LIN {X 0,Y 376.807,Z 677.795,A -85,B 0,C 180,E1 6969.755,E2 6969.755} C_VEL
LIN {X 0,Y 377.916,Z 679.038,A -85,B 0,C 180,E1 6968.251,E2 6968.251} C_VEL
LIN {X 0,Y 381.799,Z 684.185,A -85,B 0,C 180,E1 6963.881,E2 6963.881} C_VEL
LIN {X 0,Y 385.386,Z 689.219,A -85,B 0,C 180,E1 6960.565,E2 6960.565} C_VEL
LIN {X 0,Y 388.333,Z 693.407,A -85,B 0,C 180,E1 6958.19,E2 6958.19} C_VEL
LIN {X 0,Y 368.305,Z 811.662,A -85,B 0,C 180,E1 6956.59,E2 6956.59} C_VEL
LIN {X 0,Y 361.358,Z 842.659,A -85,B 0,C 180,E1 6956.015,E2 6956.015} C_VEL
LIN {X 0,Y 354.554,Z 867.168,A -85,B 0,C 180,E1 6955.437,E2 6955.437} C_VEL
LIN {X 0,Y 345.016,Z 896.006,A -85,B 0,C 180,E1 6954.606,E2 6954.606} C_VEL
LIN {X 0,Y 335.318,Z 920.733,A -85,B 0,C 180,E1 6953.73,E2 6953.73} C_VEL
LIN {X 0,Y 324.822,Z 944.388,A -85,B 0,C 180,E1 6952.726,E2 6952.726} C_VEL
LIN {X 0,Y 311.352,Z 970.875,A -85,B 0,C 180,E1 6951.358,E2 6951.358} C_VEL
LIN {X 0,Y 299.791,Z 991.138,A -85,B 0,C 180,E1 6950.092,E2 6950.092} C_VEL
LIN {X 0,Y 286.197,Z 1012.789,A -85,B 0,C 180,E1 6948.483,E2 6948.483} C_VEL
LIN {X 0,Y 270.48,Z 1035.107,A -85,B 0,C 180,E1 6946.435,E2 6946.435} C_VEL
LIN {X 0,Y 257.169,Z 1052.336,A -85,B 0,C 180,E1 6944.503,E2 6944.503} C_VEL
LIN {X 0,Y 242.609,Z 1069.728,A -85,B 0,C 180,E1 6942.133,E2 6942.133} C_VEL
LIN {X 0,Y 224.581,Z 1089.33,A -85,B 0,C 180,E1 6938.734,E2 6938.734} C_VEL
LIN {X 0,Y 210.449,Z 1103.455,A -85,B 0,C 180,E1 6935.611,E2 6935.611} C_VEL
LIN {X 0,Y 196.681,Z 1116.374,A -85,B 0,C 180,E1 6932.039,E2 6932.039} C_VEL
LIN {X 0,Y 180.199,Z 1130.963,A -85,B 0,C 180,E1 6926.819,E2 6926.819} C_VEL
LIN {X 0,Y 165.985,Z 1142.764,A -85,B 0,C 180,E1 6921.092,E2 6921.092} C_VEL
LIN {X 0,Y 154.943,Z 1151.763,A -85,B 0,C 180,E1 6915.424,E2 6915.424} C_VEL
LIN {X 0,Y 145.332,Z 1159.666,A -85,B 0,C 180,E1 6909.038,E2 6909.038} C_VEL
LIN {X 0,Y 136.611,Z 1167.272,A -85,B 0,C 180,E1 6901.115,E2 6901.115} C_VEL
LIN {X 0,Y 128.839,Z 1175.216,A -85,B 0,C 180,E1 6889.9,E2 6889.9} C_VEL
LIN {X 0,Y 125.403,Z 1180.335,A -85,B 0,C 180,E1 6880.23,E2 6880.23} C_VEL
LIN {X 0,Y 124.293,Z 1183.823,A -85,B 0,C 180,E1 6872.07,E2 6872.07} C_VEL
LIN {X 0,Y 124.366,Z 1186.875,A -85,B 0,C 180,E1 6863.576,E2 6863.576} C_VEL
LIN {X 0,Y 125.855,Z 1189.644,A -85,B 0,C 180,E1 6854.246,E2 6854.246} C_VEL
LIN {X 0,Y 129.594,Z 1191.987,A -85,B 0,C 180,E1 6844.425,E2 6844.425} C_VEL
LIN {X 0,Y 136.729,Z 1193.742,A -85,B 0,C 180,E1 6834.545,E2 6834.545} C_VEL
LIN {X 0,Y 150.578,Z 1194.995,A -85,B 0,C 180,E1 6823.409,E2 6823.409} C_VEL
LIN {X 0,Y 170.241,Z 1195.086,A -85,B 0,C 180,E1 6813.725,E2 6813.725} C_VEL
LIN {X 0,Y 142.996,Z 1208.131,A -85,B 0,C 180,E1 6799.655,E2 6799.655} C_VEL
LIN {X 0,Y 130.919,Z 1215.278,A -85,B 0,C 180,E1 6787.661,E2 6787.661} C_VEL
LIN {X 0,Y 125.246,Z 1219.957,A -85,B 0,C 180,E1 6776.555,E2 6776.555} C_VEL
LIN {X 0,Y 123.484,Z 1223.083,A -85,B 0,C 180,E1 6765.98,E2 6765.98} C_VEL
LIN {X 0,Y 123.974,Z 1224.682,A -85,B 0,C 180,E1 6757.236,E2 6757.236} C_VEL
LIN {X 0,Y 124.697,Z 1225.027,A -85,B 0,C 180,E1 6751.378,E2 6751.378} C_VEL
LIN {X 0,Y 124.597,Z 1224.748,A -85,B 0,C 180,E1 6746.78,E2 6746.78} C_VEL
LIN {X 0,Y 123.843,Z 1223.305,A -85,B 0,C 180,E1 6739.298,E2 6739.298} C_VEL
LIN {X 0,Y 124.209,Z 1220.042,A -85,B 0,C 180,E1 6729.748,E2 6729.748} C_VEL
LIN {X 0,Y 127.003,Z 1215.367,A -85,B 0,C 180,E1 6720.265,E2 6720.265} C_VEL
LIN {X 0,Y 131.824,Z 1209.964,A -85,B 0,C 180,E1 6712.078,E2 6712.078} C_VEL
LIN {X 0,Y 139.062,Z 1203.153,A -85,B 0,C 180,E1 6704.223,E2 6704.223} C_VEL
LIN {X 0,Y 148.239,Z 1195.223,A -85,B 0,C 180,E1 6697.258,E2 6697.258} C_VEL
LIN {X 0,Y 161.017,Z 1184.519,A -85,B 0,C 180,E1 6690.199,E2 6690.199} C_VEL
LIN {X 0,Y 163.262,Z 1182.63,A -85,B 0,C 180,E1 6689.177,E2 6689.177} C_VEL
LIN {X 0,Y 166.713,Z 1178.925,A -85,B 0,C 180,E1 6687.152,E2 6687.152} C_VEL
LIN {X 0,Y 173.816,Z 1168.339,A -85,B 0,C 180,E1 6681.417,E2 6681.417} C_VEL
LIN {X 0,Y 177.356,Z 1164.823,A -85,B 0,C 180,E1 6679.955,E2 6679.955} C_VEL
LIN {X 0,Y 195.152,Z 1148.924,A -85,B 0,C 180,E1 6675.148,E2 6675.148} C_VEL
LIN {X 0,Y 210.446,Z 1134.258,A -85,B 0,C 180,E1 6671.833,E2 6671.833} C_VEL
LIN {X 0,Y 226.878,Z 1117.357,A -85,B 0,C 180,E1 6668.873,E2 6668.873} C_VEL
LIN {X 0,Y 244.954,Z 1096.893,A -85,B 0,C 180,E1 6666.158,E2 6666.158} C_VEL
LIN {X 0,Y 259.21,Z 1079.289,A -85,B 0,C 180,E1 6664.338,E2 6664.338} C_VEL
LIN {X 0,Y 274.75,Z 1058.411,A -85,B 0,C 180,E1 6662.605,E2 6662.605} C_VEL
LIN {X 0,Y 290.515,Z 1034.681,A -85,B 0,C 180,E1 6661.073,E2 6661.073} C_VEL
LIN {X 0,Y 303.162,Z 1013.691,A -85,B 0,C 180,E1 6660,E2 6660} C_VEL
LIN {X 0,Y 317.013,Z 988.12,A -85,B 0,C 180,E1 6658.96,E2 6658.96} C_VEL
LIN {X 0,Y 328.622,Z 963.653,A -85,B 0,C 180,E1 6658.198,E2 6658.198} C_VEL
LIN {X 0,Y 338.703,Z 939.738,A -85,B 0,C 180,E1 6657.608,E2 6657.608} C_VEL
LIN {X 0,Y 348.992,Z 911.206,A -85,B 0,C 180,E1 6657.061,E2 6657.061} C_VEL
LIN {X 0,Y 356.194,Z 886.963,A -85,B 0,C 180,E1 6656.632,E2 6656.632} C_VEL
LIN {X 0,Y 363.113,Z 858.402,A -85,B 0,C 180,E1 6656.162,E2 6656.162} C_VEL
LIN {X 0,Y 372.946,Z 802.823,A -85,B 0,C 180,E1 6655.391,E2 6655.391} C_VEL
LIN {X 0,Y 388.709,Z 710.46,A -85,B 0,C 180,E1 6654.168,E2 6654.168} C_VEL
LIN {X 0,Y 384.521,Z 702.759,A -85,B 0,C 180,E1 6650.722,E2 6650.722} C_VEL
LIN {X 0,Y 380.976,Z 696.51,A -85,B 0,C 180,E1 6647.341,E2 6647.341} C_VEL
LIN {X 0,Y 378.128,Z 691.496,A -85,B 0,C 180,E1 6644.116,E2 6644.116} C_VEL
LIN {X 0,Y 376.181,Z 687.99,A -85,B 0,C 180,E1 6641.56,E2 6641.56} C_VEL
LIN {X 0,Y 374.754,Z 685.841,A -85,B 0,C 180,E1 6639.471,E2 6639.471} C_VEL
LIN {X 0,Y 372.295,Z 683.021,A -85,B 0,C 180,E1 6635.06,E2 6635.06} C_VEL
LIN {X 0,Y 371.245,Z 680.68,A -85,B 0,C 180,E1 6631.879,E2 6631.879} C_VEL
LIN {X 0,Y 370.079,Z 680.013,A -85,B 0,C 180,E1 6626.366,E2 6626.366} C_VEL
LIN {X 0,Y 370.244,Z 680.021,A -85,B 0,C 180,E1 6621.797,E2 6621.797} C_VEL
LIN {X 0,Y 371.851,Z 680.794,A -85,B 0,C 180,E1 6616.285,E2 6616.285} C_VEL
LIN {X 0,Y 374.459,Z 684.922,A -85,B 0,C 180,E1 6610.915,E2 6610.915} C_VEL
LIN {X 0,Y 376.119,Z 686.558,A -85,B 0,C 180,E1 6608.594,E2 6608.594} C_VEL
LIN {X 0,Y 380.047,Z 691.878,A -85,B 0,C 180,E1 6604.083,E2 6604.083} C_VEL
LIN {X 0,Y 383.547,Z 696.823,A -85,B 0,C 180,E1 6600.814,E2 6600.814} C_VEL
LIN {X 0,Y 385.447,Z 699.553,A -85,B 0,C 180,E1 6599.263,E2 6599.263} C_VEL
LIN {X 0,Y 365.956,Z 812.752,A -85,B 0,C 180,E1 6597.777,E2 6597.777} C_VEL
LIN {X 0,Y 358.945,Z 843.602,A -85,B 0,C 180,E1 6597.222,E2 6597.222} C_VEL
LIN {X 0,Y 352.057,Z 868.102,A -85,B 0,C 180,E1 6596.663,E2 6596.663} C_VEL
LIN {X 0,Y 342.867,Z 895.739,A -85,B 0,C 180,E1 6595.897,E2 6595.897} C_VEL
LIN {X 0,Y 332.641,Z 921.554,A -85,B 0,C 180,E1 6595.016,E2 6595.016} C_VEL
LIN {X 0,Y 322.146,Z 944.946,A -85,B 0,C 180,E1 6594.057,E2 6594.057} C_VEL
LIN {X 0,Y 308.801,Z 970.975,A -85,B 0,C 180,E1 6592.764,E2 6592.764} C_VEL
LIN {X 0,Y 296.588,Z 992.136,A -85,B 0,C 180,E1 6591.489,E2 6591.489} C_VEL
LIN {X 0,Y 282.347,Z 1014.496,A -85,B 0,C 180,E1 6589.875,E2 6589.875} C_VEL
LIN {X 0,Y 266.613,Z 1036.422,A -85,B 0,C 180,E1 6587.91,E2 6587.91} C_VEL
LIN {X 0,Y 253.216,Z 1053.48,A -85,B 0,C 180,E1 6586.046,E2 6586.046} C_VEL
LIN {X 0,Y 238.207,Z 1071.101,A -85,B 0,C 180,E1 6583.701,E2 6583.701} C_VEL
LIN {X 0,Y 220.296,Z 1090.178,A -85,B 0,C 180,E1 6580.46,E2 6580.46} C_VEL
LIN {X 0,Y 206.37,Z 1103.827,A -85,B 0,C 180,E1 6577.517,E2 6577.517} C_VEL
LIN {X 0,Y 192.466,Z 1116.606,A -85,B 0,C 180,E1 6574.072,E2 6574.072} C_VEL
LIN {X 0,Y 176.707,Z 1130.265,A -85,B 0,C 180,E1 6569.352,E2 6569.352} C_VEL
LIN {X 0,Y 160.645,Z 1143.256,A -85,B 0,C 180,E1 6563.209,E2 6563.209} C_VEL
LIN {X 0,Y 148.647,Z 1152.69,A -85,B 0,C 180,E1 6557.255,E2 6557.255} C_VEL
LIN {X 0,Y 138.399,Z 1160.788,A -85,B 0,C 180,E1 6550.59,E2 6550.59} C_VEL
LIN {X 0,Y 128.986,Z 1168.636,A -85,B 0,C 180,E1 6542.096,E2 6542.096} C_VEL
LIN {X 0,Y 120.895,Z 1176.564,A -85,B 0,C 180,E1 6530.281,E2 6530.281} C_VEL
LIN {X 0,Y 117.45,Z 1181.552,A -85,B 0,C 180,E1 6520.317,E2 6520.317} C_VEL
LIN {X 0,Y 116.339,Z 1185.131,A -85,B 0,C 180,E1 6511.62,E2 6511.62} C_VEL
LIN {X 0,Y 116.492,Z 1188.213,A -85,B 0,C 180,E1 6502.722,E2 6502.722} C_VEL
LIN {X 0,Y 118.291,Z 1191.127,A -85,B 0,C 180,E1 6492.696,E2 6492.696} C_VEL
LIN {X 0,Y 123.493,Z 1193.867,A -85,B 0,C 180,E1 6480.928,E2 6480.928} C_VEL
LIN {X 0,Y 132.346,Z 1195.748,A -85,B 0,C 180,E1 6470.432,E2 6470.432} C_VEL
LIN {X 0,Y 150.523,Z 1197.202,A -85,B 0,C 180,E1 6458.161,E2 6458.161} C_VEL
LIN {X 0,Y 159.73,Z 1197.368,A -85,B 0,C 180,E1 6453.838,E2 6453.838} C_VEL
LIN {X 0,Y 138.72,Z 1206.55,A -85,B 0,C 180,E1 6443.137,E2 6443.137} C_VEL
LIN {X 0,Y 125.774,Z 1213.147,A -85,B 0,C 180,E1 6431.896,E2 6431.896} C_VEL
LIN {X 0,Y 118.587,Z 1217.907,A -85,B 0,C 180,E1 6420.39,E2 6420.39} C_VEL
LIN {X 0,Y 115.75,Z 1221.168,A -85,B 0,C 180,E1 6409.163,E2 6409.163} C_VEL
LIN {X 0,Y 115.909,Z 1223.037,A -85,B 0,C 180,E1 6398.933,E2 6398.933} C_VEL
LIN {X 0,Y 116.789,Z 1223.531,A -85,B 0,C 180,E1 6391.962,E2 6391.962} C_VEL
LIN {X 0,Y 116.767,Z 1223.202,A -85,B 0,C 180,E1 6387.055,E2 6387.055} C_VEL
LIN {X 0,Y 115.963,Z 1221.726,A -85,B 0,C 180,E1 6379.065,E2 6379.065} C_VEL
LIN {X 0,Y 116.361,Z 1218.627,A -85,B 0,C 180,E1 6369.371,E2 6369.371} C_VEL
LIN {X 0,Y 119.153,Z 1214.237,A -85,B 0,C 180,E1 6359.769,E2 6359.769} C_VEL
LIN {X 0,Y 124.544,Z 1208.555,A -85,B 0,C 180,E1 6350.637,E2 6350.637} C_VEL
LIN {X 0,Y 131.983,Z 1201.99,A -85,B 0,C 180,E1 6342.705,E2 6342.705} C_VEL
LIN {X 0,Y 142.028,Z 1193.772,A -85,B 0,C 180,E1 6335.25,E2 6335.25} C_VEL
LIN {X 0,Y 156.04,Z 1182.615,A -85,B 0,C 180,E1 6327.837,E2 6327.837} C_VEL
LIN {X 0,Y 172.105,Z 1169.246,A -85,B 0,C 180,E1 6321.635,E2 6321.635} C_VEL
LIN {X 0,Y 177.356,Z 1164.823,A -85,B 0,C 180,E1 6319.955,E2 6319.955} C_VEL
LIN {X 0,Y 181.451,Z 1160.675,A -85,B 0,C 180,E1 6318.318,E2 6318.318} C_VEL
LIN {X 0,Y 190.105,Z 1148.761,A -85,B 0,C 180,E1 6313.592,E2 6313.592} C_VEL
LIN {X 0,Y 193.9,Z 1144.78,A -85,B 0,C 180,E1 6312.455,E2 6312.455} C_VEL
LIN {X 0,Y 210.652,Z 1128.923,A -85,B 0,C 180,E1 6309.146,E2 6309.146} C_VEL
LIN {X 0,Y 228.81,Z 1110.021,A -85,B 0,C 180,E1 6306.199,E2 6306.199} C_VEL
LIN {X 0,Y 243.618,Z 1093.246,A -85,B 0,C 180,E1 6304.18,E2 6304.18} C_VEL
LIN {X 0,Y 259.185,Z 1074.103,A -85,B 0,C 180,E1 6302.345,E2 6302.345} C_VEL
LIN {X 0,Y 276.159,Z 1050.89,A -85,B 0,C 180,E1 6300.622,E2 6300.622} C_VEL
LIN {X 0,Y 288.976,Z 1031.521,A -85,B 0,C 180,E1 6299.481,E2 6299.481} C_VEL
LIN {X 0,Y 302.578,Z 1008.982,A -85,B 0,C 180,E1 6298.413,E2 6298.413} C_VEL
LIN {X 0,Y 316.363,Z 983.126,A -85,B 0,C 180,E1 6297.464,E2 6297.464} C_VEL
LIN {X 0,Y 326.962,Z 960.747,A -85,B 0,C 180,E1 6296.821,E2 6296.821} C_VEL
LIN {X 0,Y 338.194,Z 933.985,A -85,B 0,C 180,E1 6296.22,E2 6296.22} C_VEL
LIN {X 0,Y 347.531,Z 907.401,A -85,B 0,C 180,E1 6295.755,E2 6295.755} C_VEL
LIN {X 0,Y 354.672,Z 883.133,A -85,B 0,C 180,E1 6295.345,E2 6295.345} C_VEL
LIN {X 0,Y 361.973,Z 851.727,A -85,B 0,C 180,E1 6294.861,E2 6294.861} C_VEL
LIN {X 0,Y 385.689,Z 715.96,A -85,B 0,C 180,E1 6293.076,E2 6293.076} C_VEL
LIN {X 0,Y 381.393,Z 708.075,A -85,B 0,C 180,E1 6289.349,E2 6289.349} C_VEL
LIN {X 0,Y 378.608,Z 703.267,A -85,B 0,C 180,E1 6286.561,E2 6286.561} C_VEL
LIN {X 0,Y 376.268,Z 699.022,A -85,B 0,C 180,E1 6283.798,E2 6283.798} C_VEL
LIN {X 0,Y 374.464,Z 695.649,A -85,B 0,C 180,E1 6281.311,E2 6281.311} C_VEL
LIN {X 0,Y 373.06,Z 693.606,A -85,B 0,C 180,E1 6279.28,E2 6279.28} C_VEL
LIN {X 0,Y 370.521,Z 690.447,A -85,B 0,C 180,E1 6274.419,E2 6274.419} C_VEL
LIN {X 0,Y 369.676,Z 688.523,A -85,B 0,C 180,E1 6271.853,E2 6271.853} C_VEL
LIN {X 0,Y 368.52,Z 687.86,A -85,B 0,C 180,E1 6266.392,E2 6266.392} C_VEL
LIN {X 0,Y 368.684,Z 687.868,A -85,B 0,C 180,E1 6261.804,E2 6261.804} C_VEL
LIN {X 0,Y 370.35,Z 688.67,A -85,B 0,C 180,E1 6256.17,E2 6256.17} C_VEL
LIN {X 0,Y 372.645,Z 692.538,A -85,B 0,C 180,E1 6251.296,E2 6251.296} C_VEL
LIN {X 0,Y 374.524,Z 694.44,A -85,B 0,C 180,E1 6248.661,E2 6248.661} C_VEL
LIN {X 0,Y 378.327,Z 699.612,A -85,B 0,C 180,E1 6244.259,E2 6244.259} C_VEL
LIN {X 0,Y 381.829,Z 704.599,A -85,B 0,C 180,E1 6240.968,E2 6240.968} C_VEL
LIN {X 0,Y 382.546,Z 705.831,A -85,B 0,C 180,E1 6240.349,E2 6240.349} C_VEL
LIN {X 0,Y 363.729,Z 813.59,A -85,B 0,C 180,E1 6238.979,E2 6238.979} C_VEL
LIN {X 0,Y 356.637,Z 844.412,A -85,B 0,C 180,E1 6238.444,E2 6238.444} C_VEL
LIN {X 0,Y 349.598,Z 869.163,A -85,B 0,C 180,E1 6237.898,E2 6237.898} C_VEL
LIN {X 0,Y 340.237,Z 896.95,A -85,B 0,C 180,E1 6237.155,E2 6237.155} C_VEL
LIN {X 0,Y 329.949,Z 922.634,A -85,B 0,C 180,E1 6236.309,E2 6236.309} C_VEL
LIN {X 0,Y 319.431,Z 945.822,A -85,B 0,C 180,E1 6235.394,E2 6235.394} C_VEL
LIN {X 0,Y 305.662,Z 972.359,A -85,B 0,C 180,E1 6234.122,E2 6234.122} C_VEL
LIN {X 0,Y 293.599,Z 993.014,A -85,B 0,C 180,E1 6232.92,E2 6232.92} C_VEL
LIN {X 0,Y 279.504,Z 1014.888,A -85,B 0,C 180,E1 6231.401,E2 6231.401} C_VEL
LIN {X 0,Y 263.536,Z 1036.941,A -85,B 0,C 180,E1 6229.504,E2 6229.504} C_VEL
LIN {X 0,Y 249.352,Z 1054.743,A -85,B 0,C 180,E1 6227.623,E2 6227.623} C_VEL
LIN {X 0,Y 233.036,Z 1073.544,A -85,B 0,C 180,E1 6225.173,E2 6225.173} C_VEL
LIN {X 0,Y 215.226,Z 1092.006,A -85,B 0,C 180,E1 6222.067,E2 6222.067} C_VEL
LIN {X 0,Y 200.472,Z 1106.103,A -85,B 0,C 180,E1 6219.045,E2 6219.045} C_VEL
LIN {X 0,Y 184.747,Z 1120.107,A -85,B 0,C 180,E1 6215.219,E2 6215.219} C_VEL
LIN {X 0,Y 166.504,Z 1135.133,A -85,B 0,C 180,E1 6209.656,E2 6209.656} C_VEL
LIN {X 0,Y 152.746,Z 1145.818,A -85,B 0,C 180,E1 6204.275,E2 6204.275} C_VEL
LIN {X 0,Y 140.894,Z 1154.778,A -85,B 0,C 180,E1 6198.339,E2 6198.339} C_VEL
LIN {X 0,Y 129.327,Z 1163.597,A -85,B 0,C 180,E1 6190.583,E2 6190.583} C_VEL
LIN {X 0,Y 118.33,Z 1172.568,A -85,B 0,C 180,E1 6179.532,E2 6179.532} C_VEL
LIN {X 0,Y 112.374,Z 1178.516,A -85,B 0,C 180,E1 6169.494,E2 6169.494} C_VEL
LIN {X 0,Y 109.356,Z 1183.037,A -85,B 0,C 180,E1 6159.795,E2 6159.795} C_VEL
LIN {X 0,Y 108.359,Z 1186.606,A -85,B 0,C 180,E1 6150.499,E2 6150.499} C_VEL
LIN {X 0,Y 108.716,Z 1189.747,A -85,B 0,C 180,E1 6141.02,E2 6141.02} C_VEL
LIN {X 0,Y 111.155,Z 1192.843,A -85,B 0,C 180,E1 6129.841,E2 6129.841} C_VEL
LIN {X 0,Y 117.496,Z 1195.665,A -85,B 0,C 180,E1 6117.561,E2 6117.561} C_VEL
LIN {X 0,Y 129.203,Z 1197.861,A -85,B 0,C 180,E1 6105.662,E2 6105.662} C_VEL
LIN {X 0,Y 149.142,Z 1199.417,A -85,B 0,C 180,E1 6093.943,E2 6093.943} C_VEL
LIN {X 0,Y 123.761,Z 1209.945,A -85,B 0,C 180,E1 6078.708,E2 6078.708} C_VEL
LIN {X 0,Y 112.841,Z 1215.61,A -85,B 0,C 180,E1 6065.391,E2 6065.391} C_VEL
LIN {X 0,Y 108.287,Z 1219.269,A -85,B 0,C 180,E1 6052.575,E2 6052.575} C_VEL
LIN {X 0,Y 107.811,Z 1221.319,A -85,B 0,C 180,E1 6041.231,E2 6041.231} C_VEL
LIN {X 0,Y 108.858,Z 1222.015,A -85,B 0,C 180,E1 6032.632,E2 6032.632} C_VEL
LIN {X 0,Y 108.975,Z 1221.736,A -85,B 0,C 180,E1 6027.897,E2 6027.897} C_VEL
LIN {X 0,Y 108.148,Z 1220.405,A -85,B 0,C 180,E1 6019.883,E2 6019.883} C_VEL
LIN {X 0,Y 108.443,Z 1217.37,A -85,B 0,C 180,E1 6009.49,E2 6009.49} C_VEL
LIN {X 0,Y 111.323,Z 1213.03,A -85,B 0,C 180,E1 5999.205,E2 5999.205} C_VEL
LIN {X 0,Y 117,Z 1207.402,A -85,B 0,C 180,E1 5989.496,E2 5989.496} C_VEL
LIN {X 0,Y 124.848,Z 1200.88,A -85,B 0,C 180,E1 5981.164,E2 5981.164} C_VEL
LIN {X 0,Y 134.856,Z 1193.116,A -85,B 0,C 180,E1 5973.786,E2 5973.786} C_VEL
LIN {X 0,Y 147.203,Z 1183.674,A -85,B 0,C 180,E1 5967.149,E2 5967.149} C_VEL
LIN {X 0,Y 165.02,Z 1169.636,A -85,B 0,C 180,E1 5960.205,E2 5960.205} C_VEL
LIN {X 0,Y 179.945,Z 1157.146,A -85,B 0,C 180,E1 5955.8,E2 5955.8} C_VEL
LIN {X 0,Y 193.9,Z 1144.78,A -85,B 0,C 180,E1 5952.455,E2 5952.455} C_VEL
LIN {X 0,Y 198.293,Z 1140.203,A -85,B 0,C 180,E1 5951.164,E2 5951.164} C_VEL
LIN {X 0,Y 207.938,Z 1127.189,A -85,B 0,C 180,E1 5947.266,E2 5947.266} C_VEL
LIN {X 0,Y 211.846,Z 1122.826,A -85,B 0,C 180,E1 5946.393,E2 5946.393} C_VEL
LIN {X 0,Y 227.953,Z 1106.085,A -85,B 0,C 180,E1 5944.024,E2 5944.024} C_VEL
LIN {X 0,Y 244.119,Z 1087.834,A -85,B 0,C 180,E1 5942.007,E2 5942.007} C_VEL
LIN {X 0,Y 261.968,Z 1065.443,A -85,B 0,C 180,E1 5940.112,E2 5940.112} C_VEL
LIN {X 0,Y 276.024,Z 1045.959,A -85,B 0,C 180,E1 5938.822,E2 5938.822} C_VEL
LIN {X 0,Y 291.219,Z 1022.84,A -85,B 0,C 180,E1 5937.603,E2 5937.603} C_VEL
LIN {X 0,Y 305.498,Z 998.135,A -85,B 0,C 180,E1 5936.604,E2 5936.604} C_VEL
LIN {X 0,Y 317.11,Z 975.773,A -85,B 0,C 180,E1 5935.891,E2 5935.891} C_VEL
LIN {X 0,Y 330.437,Z 946.425,A -85,B 0,C 180,E1 5935.177,E2 5935.177} C_VEL
LIN {X 0,Y 339.838,Z 922.429,A -85,B 0,C 180,E1 5934.742,E2 5934.742} C_VEL
LIN {X 0,Y 349.05,Z 894.753,A -85,B 0,C 180,E1 5934.288,E2 5934.288} C_VEL
LIN {X 0,Y 356.298,Z 867.232,A -85,B 0,C 180,E1 5933.866,E2 5933.866} C_VEL
LIN {X 0,Y 361.787,Z 841.172,A -85,B 0,C 180,E1 5933.497,E2 5933.497} C_VEL
LIN {X 0,Y 382.792,Z 721.682,A -85,B 0,C 180,E1 5931.983,E2 5931.983} C_VEL
LIN {X 0,Y 378.457,Z 713.573,A -85,B 0,C 180,E1 5927.953,E2 5927.953} C_VEL
LIN {X 0,Y 374.771,Z 707.129,A -85,B 0,C 180,E1 5923.89,E2 5923.89} C_VEL
LIN {X 0,Y 372.75,Z 703.307,A -85,B 0,C 180,E1 5921.06,E2 5921.06} C_VEL
LIN {X 0,Y 371.437,Z 701.418,A -85,B 0,C 180,E1 5919.186,E2 5919.186} C_VEL
LIN {X 0,Y 368.853,Z 698.114,A -85,B 0,C 180,E1 5914.123,E2 5914.123} C_VEL
LIN {X 0,Y 368.097,Z 696.361,A -85,B 0,C 180,E1 5911.793,E2 5911.793} C_VEL
LIN {X 0,Y 366.938,Z 695.699,A -85,B 0,C 180,E1 5906.212,E2 5906.212} C_VEL
LIN {X 0,Y 367.162,Z 695.714,A -85,B 0,C 180,E1 5901.617,E2 5901.617} C_VEL
LIN {X 0,Y 368.767,Z 696.511,A -85,B 0,C 180,E1 5896.257,E2 5896.257} C_VEL
LIN {X 0,Y 371.244,Z 700.558,A -85,B 0,C 180,E1 5891.084,E2 5891.084} C_VEL
LIN {X 0,Y 372.937,Z 702.331,A -85,B 0,C 180,E1 5888.72,E2 5888.72} C_VEL
LIN {X 0,Y 376.61,Z 707.346,A -85,B 0,C 180,E1 5884.437,E2 5884.437} C_VEL
LIN {X 0,Y 379.742,Z 711.795,A -85,B 0,C 180,E1 5881.455,E2 5881.455} C_VEL
LIN {X 0,Y 361.461,Z 814.915,A -85,B 0,C 180,E1 5880.185,E2 5880.185} C_VEL
LIN {X 0,Y 354.288,Z 845.626,A -85,B 0,C 180,E1 5879.668,E2 5879.668} C_VEL
LIN {X 0,Y 347.064,Z 870.673,A -85,B 0,C 180,E1 5879.136,E2 5879.136} C_VEL
LIN {X 0,Y 337.111,Z 899.588,A -85,B 0,C 180,E1 5878.384,E2 5878.384} C_VEL
LIN {X 0,Y 327.238,Z 923.891,A -85,B 0,C 180,E1 5877.611,E2 5877.611} C_VEL
LIN {X 0,Y 315.775,Z 948.792,A -85,B 0,C 180,E1 5876.66,E2 5876.66} C_VEL
LIN {X 0,Y 302.253,Z 974.281,A -85,B 0,C 180,E1 5875.471,E2 5875.471} C_VEL
LIN {X 0,Y 290.142,Z 994.707,A -85,B 0,C 180,E1 5874.321,E2 5874.321} C_VEL
LIN {X 0,Y 275.114,Z 1017.659,A -85,B 0,C 180,E1 5872.772,E2 5872.772} C_VEL
LIN {X 0,Y 259.111,Z 1039.222,A -85,B 0,C 180,E1 5870.954,E2 5870.954} C_VEL
LIN {X 0,Y 245.654,Z 1055.821,A -85,B 0,C 180,E1 5869.25,E2 5869.25} C_VEL
LIN {X 0,Y 229.617,Z 1074.022,A -85,B 0,C 180,E1 5866.963,E2 5866.963} C_VEL
LIN {X 0,Y 211.168,Z 1092.859,A -85,B 0,C 180,E1 5863.906,E2 5863.906} C_VEL
LIN {X 0,Y 196.646,Z 1106.479,A -85,B 0,C 180,E1 5861.08,E2 5861.08} C_VEL
LIN {X 0,Y 181.586,Z 1119.636,A -85,B 0,C 180,E1 5857.623,E2 5857.623} C_VEL
LIN {X 0,Y 164.164,Z 1133.873,A -85,B 0,C 180,E1 5852.692,E2 5852.692} C_VEL
LIN {X 0,Y 147.685,Z 1146.26,A -85,B 0,C 180,E1 5846.662,E2 5846.662} C_VEL
LIN {X 0,Y 135.102,Z 1155.441,A -85,B 0,C 180,E1 5840.63,E2 5840.63} C_VEL
LIN {X 0,Y 123.725,Z 1163.712,A -85,B 0,C 180,E1 5833.365,E2 5833.365} C_VEL
LIN {X 0,Y 112.42,Z 1172.473,A -85,B 0,C 180,E1 5822.802,E2 5822.802} C_VEL
LIN {X 0,Y 104.737,Z 1179.461,A -85,B 0,C 180,E1 5810.65,E2 5810.65} C_VEL
LIN {X 0,Y 101.343,Z 1184.288,A -85,B 0,C 180,E1 5799.685,E2 5799.685} C_VEL
LIN {X 0,Y 100.398,Z 1187.889,A -85,B 0,C 180,E1 5789.866,E2 5789.866} C_VEL
LIN {X 0,Y 101.043,Z 1191.256,A -85,B 0,C 180,E1 5779.06,E2 5779.06} C_VEL
LIN {X 0,Y 104.282,Z 1194.581,A -85,B 0,C 180,E1 5766.607,E2 5766.607} C_VEL
LIN {X 0,Y 111.917,Z 1197.477,A -85,B 0,C 180,E1 5753.846,E2 5753.846} C_VEL
LIN {X 0,Y 126.364,Z 1199.957,A -85,B 0,C 180,E1 5741.069,E2 5741.069} C_VEL
LIN {X 0,Y 138.626,Z 1201.05,A -85,B 0,C 180,E1 5734.068,E2 5734.068} C_VEL
LIN {X 0,Y 119.396,Z 1208.297,A -85,B 0,C 180,E1 5722.709,E2 5722.709} C_VEL
LIN {X 0,Y 107.328,Z 1213.602,A -85,B 0,C 180,E1 5710.001,E2 5710.001} C_VEL
LIN {X 0,Y 101.302,Z 1217.222,A -85,B 0,C 180,E1 5697.002,E2 5697.002} C_VEL
LIN {X 0,Y 99.773,Z 1219.484,A -85,B 0,C 180,E1 5684.509,E2 5684.509} C_VEL
LIN {X 0,Y 100.691,Z 1220.407,A -85,B 0,C 180,E1 5674.556,E2 5674.556} C_VEL
LIN {X 0,Y 101.199,Z 1220.259,A -85,B 0,C 180,E1 5669.434,E2 5669.434} C_VEL
LIN {X 0,Y 100.547,Z 1219.543,A -85,B 0,C 180,E1 5663.146,E2 5663.146} C_VEL
LIN {X 0,Y 100.279,Z 1216.913,A -85,B 0,C 180,E1 5651.995,E2 5651.995} C_VEL
LIN {X 0,Y 103.504,Z 1211.835,A -85,B 0,C 180,E1 5638.557,E2 5638.557} C_VEL
LIN {X 0,Y 109.509,Z 1206.248,A -85,B 0,C 180,E1 5628.2,E2 5628.2} C_VEL
LIN {X 0,Y 117.815,Z 1199.764,A -85,B 0,C 180,E1 5619.439,E2 5619.439} C_VEL
LIN {X 0,Y 128.292,Z 1192.078,A -85,B 0,C 180,E1 5611.841,E2 5611.841} C_VEL
LIN {X 0,Y 141.27,Z 1182.624,A -85,B 0,C 180,E1 5605.048,E2 5605.048} C_VEL
LIN {X 0,Y 159.054,Z 1169.201,A -85,B 0,C 180,E1 5598.32,E2 5598.32} C_VEL
LIN {X 0,Y 175.014,Z 1156.289,A -85,B 0,C 180,E1 5593.777,E2 5593.777} C_VEL
LIN {X 0,Y 190.067,Z 1143.312,A -85,B 0,C 180,E1 5590.346,E2 5590.346} C_VEL
LIN {X 0,Y 208.499,Z 1126.22,A -85,B 0,C 180,E1 5586.934,E2 5586.934} C_VEL
LIN {X 0,Y 211.846,Z 1122.826,A -85,B 0,C 180,E1 5586.393,E2 5586.393} C_VEL
LIN {X 0,Y 216.307,Z 1117.758,A -85,B 0,C 180,E1 5585.4,E2 5585.4} C_VEL
LIN {X 0,Y 226.31,Z 1103.662,A -85,B 0,C 180,E1 5582.194,E2 5582.194} C_VEL
LIN {X 0,Y 230.269,Z 1099.009,A -85,B 0,C 180,E1 5581.498,E2 5581.498} C_VEL
LIN {X 0,Y 248.072,Z 1078.27,A -85,B 0,C 180,E1 5579.538,E2 5579.538} C_VEL
LIN {X 0,Y 262.602,Z 1059.728,A -85,B 0,C 180,E1 5578.162,E2 5578.162} C_VEL
LIN {X 0,Y 279.407,Z 1036.037,A -85,B 0,C 180,E1 5576.777,E2 5576.777} C_VEL
LIN {X 0,Y 293.253,Z 1014.098,A -85,B 0,C 180,E1 5575.794,E2 5575.794} C_VEL
LIN {X 0,Y 305.617,Z 992.449,A -85,B 0,C 180,E1 5575.018,E2 5575.018} C_VEL
LIN {X 0,Y 319.647,Z 964.658,A -85,B 0,C 180,E1 5574.255,E2 5574.255} C_VEL
LIN {X 0,Y 329.909,Z 941.343,A -85,B 0,C 180,E1 5573.768,E2 5573.768} C_VEL
LIN {X 0,Y 340.26,Z 914.537,A -85,B 0,C 180,E1 5573.331,E2 5573.331} C_VEL
LIN {X 0,Y 348.971,Z 886.699,A -85,B 0,C 180,E1 5572.911,E2 5572.911} C_VEL
LIN {X 0,Y 355.409,Z 861.609,A -85,B 0,C 180,E1 5572.546,E2 5572.546} C_VEL
LIN {X 0,Y 362.892,Z 823.483,A -85,B 0,C 180,E1 5572.051,E2 5572.051} C_VEL
LIN {X 0,Y 379.925,Z 727.388,A -85,B 0,C 180,E1 5570.876,E2 5570.876} C_VEL
LIN {X 0,Y 375.982,Z 720.12,A -85,B 0,C 180,E1 5567.092,E2 5567.092} C_VEL
LIN {X 0,Y 372.918,Z 714.656,A -85,B 0,C 180,E1 5563.568,E2 5563.568} C_VEL
LIN {X 0,Y 370.981,Z 710.947,A -85,B 0,C 180,E1 5560.803,E2 5560.803} C_VEL
LIN {X 0,Y 369.816,Z 709.23,A -85,B 0,C 180,E1 5559.09,E2 5559.09} C_VEL
LIN {X 0,Y 367.211,Z 705.883,A -85,B 0,C 180,E1 5553.969,E2 5553.969} C_VEL
LIN {X 0,Y 366.495,Z 704.188,A -85,B 0,C 180,E1 5551.659,E2 5551.659} C_VEL
LIN {X 0,Y 365.378,Z 703.546,A -85,B 0,C 180,E1 5546.253,E2 5546.253} C_VEL
LIN {X 0,Y 365.596,Z 703.56,A -85,B 0,C 180,E1 5541.622,E2 5541.622} C_VEL
LIN {X 0,Y 367.208,Z 704.449,A -85,B 0,C 180,E1 5536.24,E2 5536.24} C_VEL
LIN {X 0,Y 369.743,Z 708.477,A -85,B 0,C 180,E1 5531.018,E2 5531.018} C_VEL
LIN {X 0,Y 371.294,Z 710.117,A -85,B 0,C 180,E1 5528.863,E2 5528.863} C_VEL
LIN {X 0,Y 374.897,Z 715.08,A -85,B 0,C 180,E1 5524.617,E2 5524.617} C_VEL
LIN {X 0,Y 376.988,Z 718.191,A -85,B 0,C 180,E1 5522.564,E2 5522.564} C_VEL
LIN {X 0,Y 359.439,Z 815.795,A -85,B 0,C 180,E1 5521.41,E2 5521.41} C_VEL
LIN {X 0,Y 352.188,Z 846.506,A -85,B 0,C 180,E1 5520.915,E2 5520.915} C_VEL
LIN {X 0,Y 345.103,Z 870.856,A -85,B 0,C 180,E1 5520.42,E2 5520.42} C_VEL
LIN {X 0,Y 335.312,Z 899.261,A -85,B 0,C 180,E1 5519.72,E2 5519.72} C_VEL
LIN {X 0,Y 325.051,Z 924.337,A -85,B 0,C 180,E1 5518.961,E2 5518.961} C_VEL
LIN {X 0,Y 314.124,Z 947.918,A -85,B 0,C 180,E1 5518.105,E2 5518.105} C_VEL
LIN {X 0,Y 299.898,Z 974.682,A -85,B 0,C 180,E1 5516.924,E2 5516.924} C_VEL
LIN {X 0,Y 287.264,Z 995.772,A -85,B 0,C 180,E1 5515.791,E2 5515.791} C_VEL
LIN {X 0,Y 272.05,Z 1018.717,A -85,B 0,C 180,E1 5514.308,E2 5514.308} C_VEL
LIN {X 0,Y 256.036,Z 1040.031,A -85,B 0,C 180,E1 5512.588,E2 5512.588} C_VEL
LIN {X 0,Y 241.58,Z 1057.601,A -85,B 0,C 180,E1 5510.851,E2 5510.851} C_VEL
LIN {X 0,Y 224.113,Z 1077.023,A -85,B 0,C 180,E1 5508.467,E2 5508.467} C_VEL
LIN {X 0,Y 206.221,Z 1094.775,A -85,B 0,C 180,E1 5505.625,E2 5505.625} C_VEL
LIN {X 0,Y 190.718,Z 1108.961,A -85,B 0,C 180,E1 5502.72,E2 5502.72} C_VEL
LIN {X 0,Y 172.759,Z 1124.191,A -85,B 0,C 180,E1 5498.655,E2 5498.655} C_VEL
LIN {X 0,Y 154.719,Z 1138.077,A -85,B 0,C 180,E1 5493.479,E2 5493.479} C_VEL
LIN {X 0,Y 140.066,Z 1148.7,A -85,B 0,C 180,E1 5488.059,E2 5488.059} C_VEL
LIN {X 0,Y 126.31,Z 1158.329,A -85,B 0,C 180,E1 5481.35,E2 5481.35} C_VEL
LIN {X 0,Y 111.061,Z 1169.013,A -85,B 0,C 180,E1 5470.543,E2 5470.543} C_VEL
LIN {X 0,Y 102.119,Z 1175.79,A -85,B 0,C 180,E1 5460.627,E2 5460.627} C_VEL
LIN {X 0,Y 96.25,Z 1181.322,A -85,B 0,C 180,E1 5449.904,E2 5449.904} C_VEL
LIN {X 0,Y 93.275,Z 1185.661,A -85,B 0,C 180,E1 5439.233,E2 5439.233} C_VEL
LIN {X 0,Y 92.42,Z 1189.334,A -85,B 0,C 180,E1 5428.427,E2 5428.427} C_VEL
LIN {X 0,Y 93.417,Z 1192.776,A -85,B 0,C 180,E1 5416.798,E2 5416.798} C_VEL
LIN {X 0,Y 97.703,Z 1196.328,A -85,B 0,C 180,E1 5402.933,E2 5402.933} C_VEL
LIN {X 0,Y 106.802,Z 1199.317,A -85,B 0,C 180,E1 5389.754,E2 5389.754} C_VEL
LIN {X 0,Y 123.077,Z 1201.92,A -85,B 0,C 180,E1 5377.048,E2 5377.048} C_VEL
LIN {X 0,Y 128.006,Z 1202.581,A -85,B 0,C 180,E1 5374.188,E2 5374.188} C_VEL
LIN {X 0,Y 105.018,Z 1210.615,A -85,B 0,C 180,E1 5357.956,E2 5357.956} C_VEL
LIN {X 0,Y 95.048,Z 1215.079,A -85,B 0,C 180,E1 5342.446,E2 5342.446} C_VEL
LIN {X 0,Y 91.952,Z 1217.683,A -85,B 0,C 180,E1 5327.726,E2 5327.726} C_VEL
LIN {X 0,Y 92.58,Z 1218.777,A -85,B 0,C 180,E1 5316.2,E2 5316.2} C_VEL
LIN {X 0,Y 93.34,Z 1218.727,A -85,B 0,C 180,E1 5310.614,E2 5310.614} C_VEL
LIN {X 0,Y 92.979,Z 1218.301,A -85,B 0,C 180,E1 5305.683,E2 5305.683} C_VEL
LIN {X 0,Y 92.271,Z 1216.317,A -85,B 0,C 180,E1 5295.568,E2 5295.568} C_VEL
LIN {X 0,Y 93.824,Z 1212.734,A -85,B 0,C 180,E1 5283.411,E2 5283.411} C_VEL
LIN {X 0,Y 100.487,Z 1206.358,A -85,B 0,C 180,E1 5268.95,E2 5268.95} C_VEL
LIN {X 0,Y 110.353,Z 1198.978,A -85,B 0,C 180,E1 5257.975,E2 5257.975} C_VEL
LIN {X 0,Y 121.297,Z 1191.389,A -85,B 0,C 180,E1 5250.056,E2 5250.056} C_VEL
LIN {X 0,Y 134.036,Z 1182.547,A -85,B 0,C 180,E1 5243.429,E2 5243.429} C_VEL
LIN {X 0,Y 149.013,Z 1171.828,A -85,B 0,C 180,E1 5237.67,E2 5237.67} C_VEL
LIN {X 0,Y 168.69,Z 1156.67,A -85,B 0,C 180,E1 5232.039,E2 5232.039} C_VEL
LIN {X 0,Y 184.065,Z 1143.85,A -85,B 0,C 180,E1 5228.637,E2 5228.637} C_VEL
LIN {X 0,Y 199.034,Z 1130.446,A -85,B 0,C 180,E1 5225.911,E2 5225.911} C_VEL
LIN {X 0,Y 217.301,Z 1112.737,A -85,B 0,C 180,E1 5223.149,E2 5223.149} C_VEL
LIN {X 0,Y 230.269,Z 1099.009,A -85,B 0,C 180,E1 5221.498,E2 5221.498} C_VEL
LIN {X 0,Y 234.758,Z 1093.557,A -85,B 0,C 180,E1 5220.703,E2 5220.703} C_VEL
LIN {X 0,Y 244.623,Z 1078.354,A -85,B 0,C 180,E1 5218.047,E2 5218.047} C_VEL
LIN {X 0,Y 248.387,Z 1073.371,A -85,B 0,C 180,E1 5217.506,E2 5217.506} C_VEL
LIN {X 0,Y 266.624,Z 1049.674,A -85,B 0,C 180,E1 5215.975,E2 5215.975} C_VEL
LIN {X 0,Y 281.065,Z 1028.644,A -85,B 0,C 180,E1 5214.93,E2 5214.93} C_VEL
LIN {X 0,Y 295.055,Z 1006.159,A -85,B 0,C 180,E1 5214.047,E2 5214.047} C_VEL
LIN {X 0,Y 309.086,Z 980.596,A -85,B 0,C 180,E1 5213.279,E2 5213.279} C_VEL
LIN {X 0,Y 320.013,Z 958.14,A -85,B 0,C 180,E1 5212.758,E2 5212.758} C_VEL
LIN {X 0,Y 331.46,Z 931.575,A -85,B 0,C 180,E1 5212.284,E2 5212.284} C_VEL
LIN {X 0,Y 341.046,Z 904.961,A -85,B 0,C 180,E1 5211.91,E2 5211.91} C_VEL
LIN {X 0,Y 348.471,Z 880.415,A -85,B 0,C 180,E1 5211.559,E2 5211.559} C_VEL
LIN {X 0,Y 355.992,Z 849.08,A -85,B 0,C 180,E1 5211.136,E2 5211.136} C_VEL
LIN {X 0,Y 377.049,Z 733.269,A -85,B 0,C 180,E1 5209.765,E2 5209.765} C_VEL
LIN {X 0,Y 373.766,Z 727.148,A -85,B 0,C 180,E1 5206.463,E2 5206.463} C_VEL
LIN {X 0,Y 371.124,Z 722.293,A -85,B 0,C 180,E1 5203.325,E2 5203.325} C_VEL
LIN {X 0,Y 369.323,Z 718.773,A -85,B 0,C 180,E1 5200.713,E2 5200.713} C_VEL
LIN {X 0,Y 368.181,Z 717.039,A -85,B 0,C 180,E1 5198.993,E2 5198.993} C_VEL
LIN {X 0,Y 365.511,Z 713.556,A -85,B 0,C 180,E1 5193.694,E2 5193.694} C_VEL
LIN {X 0,Y 364.882,Z 712.012,A -85,B 0,C 180,E1 5191.522,E2 5191.522} C_VEL
LIN {X 0,Y 363.788,Z 711.383,A -85,B 0,C 180,E1 5186.085,E2 5186.085} C_VEL
LIN {X 0,Y 364.064,Z 711.43,A -85,B 0,C 180,E1 5181.431,E2 5181.431} C_VEL
LIN {X 0,Y 365.599,Z 712.19,A -85,B 0,C 180,E1 5176.433,E2 5176.433} C_VEL
LIN {X 0,Y 368.221,Z 716.374,A -85,B 0,C 180,E1 5170.983,E2 5170.983} C_VEL
LIN {X 0,Y 369.675,Z 717.94,A -85,B 0,C 180,E1 5168.976,E2 5168.976} C_VEL
LIN {X 0,Y 373.091,Z 722.649,A -85,B 0,C 180,E1 5164.906,E2 5164.906} C_VEL
LIN {X 0,Y 374.256,Z 724.516,A -85,B 0,C 180,E1 5163.69,E2 5163.69} C_VEL
LIN {X 0,Y 357.405,Z 816.99,A -85,B 0,C 180,E1 5162.642,E2 5162.642} C_VEL
LIN {X 0,Y 350.081,Z 847.572,A -85,B 0,C 180,E1 5162.167,E2 5162.167} C_VEL
LIN {X 0,Y 342.697,Z 872.627,A -85,B 0,C 180,E1 5161.68,E2 5161.68} C_VEL
LIN {X 0,Y 332.23,Z 902.302,A -85,B 0,C 180,E1 5160.973,E2 5160.973} C_VEL
LIN {X 0,Y 322.038,Z 926.807,A -85,B 0,C 180,E1 5160.257,E2 5160.257} C_VEL
LIN {X 0,Y 309.706,Z 952.901,A -85,B 0,C 180,E1 5159.343,E2 5159.343} C_VEL
LIN {X 0,Y 296.383,Z 977.222,A -85,B 0,C 180,E1 5158.294,E2 5158.294} C_VEL
LIN {X 0,Y 283.611,Z 998.2,A -85,B 0,C 180,E1 5157.208,E2 5157.208} C_VEL
LIN {X 0,Y 266.632,Z 1023.064,A -85,B 0,C 180,E1 5155.639,E2 5155.639} C_VEL
LIN {X 0,Y 251.927,Z 1042.271,A -85,B 0,C 180,E1 5154.129,E2 5154.129} C_VEL
LIN {X 0,Y 236.862,Z 1060.232,A -85,B 0,C 180,E1 5152.408,E2 5152.408} C_VEL
LIN {X 0,Y 217.535,Z 1081.001,A -85,B 0,C 180,E1 5149.885,E2 5149.885} C_VEL
LIN {X 0,Y 201.69,Z 1096.381,A -85,B 0,C 180,E1 5147.466,E2 5147.466} C_VEL
LIN {X 0,Y 185.864,Z 1110.534,A -85,B 0,C 180,E1 5144.646,E2 5144.646} C_VEL
LIN {X 0,Y 166.776,Z 1126.26,A -85,B 0,C 180,E1 5140.501,E2 5140.501} C_VEL
LIN {X 0,Y 149.549,Z 1139.114,A -85,B 0,C 180,E1 5135.756,E2 5135.756} C_VEL
LIN {X 0,Y 134.994,Z 1149.343,A -85,B 0,C 180,E1 5130.627,E2 5130.627} C_VEL
LIN {X 0,Y 121.322,Z 1158.57,A -85,B 0,C 180,E1 5124.324,E2 5124.324} C_VEL
LIN {X 0,Y 106.714,Z 1168.396,A -85,B 0,C 180,E1 5114.791,E2 5114.791} C_VEL
LIN {X 0,Y 94.733,Z 1176.841,A -85,B 0,C 180,E1 5102.328,E2 5102.328} C_VEL
LIN {X 0,Y 88.263,Z 1182.584,A -85,B 0,C 180,E1 5090.385,E2 5090.385} C_VEL
LIN {X 0,Y 85.18,Z 1187.065,A -85,B 0,C 180,E1 5078.474,E2 5078.474} C_VEL
LIN {X 0,Y 84.508,Z 1190.786,A -85,B 0,C 180,E1 5066.719,E2 5066.719} C_VEL
LIN {X 0,Y 85.914,Z 1194.277,A -85,B 0,C 180,E1 5054.147,E2 5054.147} C_VEL
LIN {X 0,Y 91.562,Z 1198.059,A -85,B 0,C 180,E1 5038.749,E2 5038.749} C_VEL
LIN {X 0,Y 102.808,Z 1201.269,A -85,B 0,C 180,E1 5024.776,E2 5024.776} C_VEL
LIN {X 0,Y 117.454,Z 1203.582,A -85,B 0,C 180,E1 5014.331,E2 5014.331} C_VEL
LIN {X 0,Y 98.977,Z 1209.448,A -85,B 0,C 180,E1 5001.065,E2 5001.065} C_VEL
LIN {X 0,Y 88.685,Z 1213.313,A -85,B 0,C 180,E1 4986.694,E2 4986.694} C_VEL
LIN {X 0,Y 84.347,Z 1215.848,A -85,B 0,C 180,E1 4971.56,E2 4971.56} C_VEL
LIN {X 0,Y 84.564,Z 1217.095,A -85,B 0,C 180,E1 4957.473,E2 4957.473} C_VEL
LIN {X 0,Y 85.499,Z 1217.092,A -85,B 0,C 180,E1 4950.67,E2 4950.67} C_VEL
LIN {X 0,Y 85.136,Z 1216.732,A -85,B 0,C 180,E1 4945.959,E2 4945.959} C_VEL
LIN {X 0,Y 84.424,Z 1214.677,A -85,B 0,C 180,E1 4934.897,E2 4934.897} C_VEL
LIN {X 0,Y 86.953,Z 1210.361,A -85,B 0,C 180,E1 4919.592,E2 4919.592} C_VEL
LIN {X 0,Y 94.312,Z 1204.131,A -85,B 0,C 180,E1 4905.595,E2 4905.595} C_VEL
LIN {X 0,Y 104.145,Z 1197.381,A -85,B 0,C 180,E1 4895.307,E2 4895.307} C_VEL
LIN {X 0,Y 115.84,Z 1189.742,A -85,B 0,C 180,E1 4887.225,E2 4887.225} C_VEL
LIN {X 0,Y 129.269,Z 1180.87,A -85,B 0,C 180,E1 4880.623,E2 4880.623} C_VEL
LIN {X 0,Y 146.615,Z 1168.926,A -85,B 0,C 180,E1 4874.441,E2 4874.441} C_VEL
LIN {X 0,Y 165.261,Z 1154.819,A -85,B 0,C 180,E1 4869.531,E2 4869.531} C_VEL
LIN {X 0,Y 181.064,Z 1141.94,A -85,B 0,C 180,E1 4866.281,E2 4866.281} C_VEL
LIN {X 0,Y 197.77,Z 1127.213,A -85,B 0,C 180,E1 4863.478,E2 4863.478} C_VEL
LIN {X 0,Y 217.99,Z 1107.505,A -85,B 0,C 180,E1 4860.716,E2 4860.716} C_VEL
LIN {X 0,Y 233.509,Z 1090.807,A -85,B 0,C 180,E1 4858.96,E2 4858.96} C_VEL
LIN {X 0,Y 248.387,Z 1073.371,A -85,B 0,C 180,E1 4857.506,E2 4857.506} C_VEL
LIN {X 0,Y 252.723,Z 1067.537,A -85,B 0,C 180,E1 4856.875,E2 4856.875} C_VEL
LIN {X 0,Y 262.401,Z 1051.567,A -85,B 0,C 180,E1 4854.632,E2 4854.632} C_VEL
LIN {X 0,Y 265.918,Z 1046.218,A -85,B 0,C 180,E1 4854.209,E2 4854.209} C_VEL
LIN {X 0,Y 279.878,Z 1025.954,A -85,B 0,C 180,E1 4853.298,E2 4853.298} C_VEL
LIN {X 0,Y 295.404,Z 1000.864,A -85,B 0,C 180,E1 4852.414,E2 4852.414} C_VEL
LIN {X 0,Y 308.164,Z 977.389,A -85,B 0,C 180,E1 4851.792,E2 4851.792} C_VEL
LIN {X 0,Y 319.633,Z 953.714,A -85,B 0,C 180,E1 4851.306,E2 4851.306} C_VEL
LIN {X 0,Y 331.507,Z 925.383,A -85,B 0,C 180,E1 4850.875,E2 4850.875} C_VEL
LIN {X 0,Y 339.99,Z 901.544,A -85,B 0,C 180,E1 4850.567,E2 4850.567} C_VEL
LIN {X 0,Y 348.431,Z 873.126,A -85,B 0,C 180,E1 4850.186,E2 4850.186} C_VEL
LIN {X 0,Y 354.916,Z 844.792,A -85,B 0,C 180,E1 4849.832,E2 4849.832} C_VEL
LIN {X 0,Y 374.342,Z 739.107,A -85,B 0,C 180,E1 4848.65,E2 4848.65} C_VEL
LIN {X 0,Y 371.189,Z 733.377,A -85,B 0,C 180,E1 4845.332,E2 4845.332} C_VEL
LIN {X 0,Y 368.185,Z 727.359,A -85,B 0,C 180,E1 4841.309,E2 4841.309} C_VEL
LIN {X 0,Y 366.542,Z 724.845,A -85,B 0,C 180,E1 4838.895,E2 4838.895} C_VEL
LIN {X 0,Y 363.742,Z 721.061,A -85,B 0,C 180,E1 4833.203,E2 4833.203} C_VEL
LIN {X 0,Y 363.268,Z 719.835,A -85,B 0,C 180,E1 4831.384,E2 4831.384} C_VEL
LIN {X 0,Y 362.201,Z 719.219,A -85,B 0,C 180,E1 4825.911,E2 4825.911} C_VEL
LIN {X 0,Y 362.536,Z 719.301,A -85,B 0,C 180,E1 4821.238,E2 4821.238} C_VEL
LIN {X 0,Y 364.032,Z 720.124,A -85,B 0,C 180,E1 4816.415,E2 4816.415} C_VEL
LIN {X 0,Y 366.699,Z 724.271,A -85,B 0,C 180,E1 4810.948,E2 4810.948} C_VEL
LIN {X 0,Y 368.058,Z 725.785,A -85,B 0,C 180,E1 4809.069,E2 4809.069} C_VEL
LIN {X 0,Y 371.482,Z 730.546,A -85,B 0,C 180,E1 4804.981,E2 4804.981} C_VEL
LIN {X 0,Y 371.576,Z 730.994,A -85,B 0,C 180,E1 4804.828,E2 4804.828} C_VEL
LIN {X 0,Y 355.396,Z 818.451,A -85,B 0,C 180,E1 4803.881,E2 4803.881} C_VEL
LIN {X 0,Y 348.033,Z 848.777,A -85,B 0,C 180,E1 4803.43,E2 4803.43} C_VEL
LIN {X 0,Y 340.555,Z 873.854,A -85,B 0,C 180,E1 4802.966,E2 4802.966} C_VEL
LIN {X 0,Y 330.031,Z 903.368,A -85,B 0,C 180,E1 4802.297,E2 4802.297} C_VEL
LIN {X 0,Y 319.89,Z 927.533,A -85,B 0,C 180,E1 4801.628,E2 4801.628} C_VEL
LIN {X 0,Y 307.718,Z 953.106,A -85,B 0,C 180,E1 4800.781,E2 4800.781} C_VEL
LIN {X 0,Y 294.005,Z 977.976,A -85,B 0,C 180,E1 4799.771,E2 4799.771} C_VEL
LIN {X 0,Y 281.473,Z 998.396,A -85,B 0,C 180,E1 4798.773,E2 4798.773} C_VEL
LIN {X 0,Y 265.277,Z 1022.103,A -85,B 0,C 180,E1 4797.377,E2 4797.377} C_VEL
LIN {X 0,Y 249.635,Z 1042.387,A -85,B 0,C 180,E1 4795.886,E2 4795.886} C_VEL
LIN {X 0,Y 234.797,Z 1059.941,A -85,B 0,C 180,E1 4794.31,E2 4794.31} C_VEL
LIN {X 0,Y 216.607,Z 1079.529,A -85,B 0,C 180,E1 4792.114,E2 4792.114} C_VEL
LIN {X 0,Y 198.421,Z 1096.967,A -85,B 0,C 180,E1 4789.551,E2 4789.551} C_VEL
LIN {X 0,Y 182.964,Z 1110.599,A -85,B 0,C 180,E1 4786.986,E2 4786.986} C_VEL
LIN {X 0,Y 165.578,Z 1124.739,A -85,B 0,C 180,E1 4783.529,E2 4783.529} C_VEL
LIN {X 0,Y 145.082,Z 1139.854,A -85,B 0,C 180,E1 4778.322,E2 4778.322} C_VEL
LIN {X 0,Y 129.162,Z 1150.706,A -85,B 0,C 180,E1 4772.989,E2 4772.989} C_VEL
LIN {X 0,Y 114.229,Z 1160.362,A -85,B 0,C 180,E1 4766.279,E2 4766.279} C_VEL
LIN {X 0,Y 98.074,Z 1170.683,A -85,B 0,C 180,E1 4755.594,E2 4755.594} C_VEL
LIN {X 0,Y 86.464,Z 1178.521,A -85,B 0,C 180,E1 4742.93,E2 4742.93} C_VEL
LIN {X 0,Y 80.087,Z 1184.047,A -85,B 0,C 180,E1 4730.452,E2 4730.452} C_VEL
LIN {X 0,Y 77.091,Z 1188.458,A -85,B 0,C 180,E1 4717.561,E2 4717.561} C_VEL
LIN {X 0,Y 76.631,Z 1192.205,A -85,B 0,C 180,E1 4704.68,E2 4704.68} C_VEL
LIN {X 0,Y 78.584,Z 1195.775,A -85,B 0,C 180,E1 4691.003,E2 4691.003} C_VEL
LIN {X 0,Y 86.816,Z 1200.078,A -85,B 0,C 180,E1 4672.722,E2 4672.722} C_VEL
LIN {X 0,Y 102.217,Z 1203.67,A -85,B 0,C 180,E1 4657.573,E2 4657.573} C_VEL
LIN {X 0,Y 106.877,Z 1204.474,A -85,B 0,C 180,E1 4654.51,E2 4654.51} C_VEL
LIN {X 0,Y 85.855,Z 1210.557,A -85,B 0,C 180,E1 4636.224,E2 4636.224} C_VEL
LIN {X 0,Y 77.634,Z 1213.706,A -85,B 0,C 180,E1 4618.459,E2 4618.459} C_VEL
LIN {X 0,Y 76.248,Z 1215.269,A -85,B 0,C 180,E1 4602.111,E2 4602.111} C_VEL
LIN {X 0,Y 77.579,Z 1215.478,A -85,B 0,C 180,E1 4591.477,E2 4591.477} C_VEL
LIN {X 0,Y 77.403,Z 1215.224,A -85,B 0,C 180,E1 4587.038,E2 4587.038} C_VEL
LIN {X 0,Y 76.566,Z 1213.166,A -85,B 0,C 180,E1 4574.86,E2 4574.86} C_VEL
LIN {X 0,Y 79.393,Z 1208.766,A -85,B 0,C 180,E1 4558.065,E2 4558.065} C_VEL
LIN {X 0,Y 87.147,Z 1202.769,A -85,B 0,C 180,E1 4543.505,E2 4543.505} C_VEL
LIN {X 0,Y 97.561,Z 1196.127,A -85,B 0,C 180,E1 4532.818,E2 4532.818} C_VEL
LIN {X 0,Y 109.924,Z 1188.525,A -85,B 0,C 180,E1 4524.549,E2 4524.549} C_VEL
LIN {X 0,Y 124.396,Z 1179.426,A -85,B 0,C 180,E1 4517.785,E2 4517.785} C_VEL
LIN {X 0,Y 142.909,Z 1167.115,A -85,B 0,C 180,E1 4511.614,E2 4511.614} C_VEL
LIN {X 0,Y 161.225,Z 1153.658,A -85,B 0,C 180,E1 4507.123,E2 4507.123} C_VEL
LIN {X 0,Y 177.414,Z 1140.787,A -85,B 0,C 180,E1 4504.016,E2 4504.016} C_VEL
LIN {X 0,Y 194.035,Z 1126.442,A -85,B 0,C 180,E1 4501.418,E2 4501.418} C_VEL
LIN {X 0,Y 215.024,Z 1106.363,A -85,B 0,C 180,E1 4498.756,E2 4498.756} C_VEL
LIN {X 0,Y 231.276,Z 1089.101,A -85,B 0,C 180,E1 4497.059,E2 4497.059} C_VEL
LIN {X 0,Y 247.702,Z 1069.992,A -85,B 0,C 180,E1 4495.593,E2 4495.593} C_VEL
LIN {X 0,Y 265.633,Z 1046.616,A -85,B 0,C 180,E1 4494.229,E2 4494.229} C_VEL
LIN {X 0,Y 265.918,Z 1046.218,A -85,B 0,C 180,E1 4494.209,E2 4494.209} C_VEL
LIN {X 0,Y 269.965,Z 1040.021,A -85,B 0,C 180,E1 4493.709,E2 4493.709} C_VEL
LIN {X 0,Y 279.192,Z 1023.211,A -85,B 0,C 180,E1 4491.794,E2 4491.794} C_VEL
LIN {X 0,Y 282.446,Z 1017.638,A -85,B 0,C 180,E1 4491.46,E2 4491.46} C_VEL
LIN {X 0,Y 296.82,Z 993.559,A -85,B 0,C 180,E1 4490.754,E2 4490.754} C_VEL
LIN {X 0,Y 308.932,Z 970.928,A -85,B 0,C 180,E1 4490.241,E2 4490.241} C_VEL
LIN {X 0,Y 322.087,Z 942.764,A -85,B 0,C 180,E1 4489.764,E2 4489.764} C_VEL
LIN {X 0,Y 331.537,Z 919.405,A -85,B 0,C 180,E1 4489.476,E2 4489.476} C_VEL
LIN {X 0,Y 340.747,Z 892.83,A -85,B 0,C 180,E1 4489.152,E2 4489.152} C_VEL
LIN {X 0,Y 348.589,Z 864.402,A -85,B 0,C 180,E1 4488.806,E2 4488.806} C_VEL
LIN {X 0,Y 354.276,Z 838.711,A -85,B 0,C 180,E1 4488.505,E2 4488.505} C_VEL
LIN {X 0,Y 371.603,Z 745.1,A -85,B 0,C 180,E1 4487.53,E2 4487.53} C_VEL
LIN {X 0,Y 367.879,Z 738.141,A -85,B 0,C 180,E1 4483.255,E2 4483.255} C_VEL
LIN {X 0,Y 365.88,Z 734.231,A -85,B 0,C 180,E1 4480.358,E2 4480.358} C_VEL
LIN {X 0,Y 364.794,Z 732.567,A -85,B 0,C 180,E1 4478.62,E2 4478.62} C_VEL
LIN {X 0,Y 362.11,Z 728.849,A -85,B 0,C 180,E1 4473.073,E2 4473.073} C_VEL
LIN {X 0,Y 361.656,Z 727.658,A -85,B 0,C 180,E1 4471.245,E2 4471.245} C_VEL
LIN {X 0,Y 360.629,Z 727.064,A -85,B 0,C 180,E1 4465.939,E2 4465.939} C_VEL
LIN {X 0,Y 360.966,Z 727.145,A -85,B 0,C 180,E1 4461.242,E2 4461.242} C_VEL
LIN {X 0,Y 362.465,Z 728.055,A -85,B 0,C 180,E1 4456.398,E2 4456.398} C_VEL
LIN {X 0,Y 365.207,Z 732.195,A -85,B 0,C 180,E1 4450.87,E2 4450.87} C_VEL
LIN {X 0,Y 366.414,Z 733.588,A -85,B 0,C 180,E1 4449.195,E2 4449.195} C_VEL
LIN {X 0,Y 369.02,Z 737.242,A -85,B 0,C 180,E1 4445.983,E2 4445.983} C_VEL
LIN {X 0,Y 353.709,Z 819.153,A -85,B 0,C 180,E1 4445.141,E2 4445.141} C_VEL
LIN {X 0,Y 346.319,Z 849.376,A -85,B 0,C 180,E1 4444.716,E2 4444.716} C_VEL
LIN {X 0,Y 338.833,Z 874.309,A -85,B 0,C 180,E1 4444.281,E2 4444.281} C_VEL
LIN {X 0,Y 328.341,Z 903.619,A -85,B 0,C 180,E1 4443.658,E2 4443.658} C_VEL
LIN {X 0,Y 317.956,Z 928.197,A -85,B 0,C 180,E1 4443.018,E2 4443.018} C_VEL
LIN {X 0,Y 305.67,Z 953.806,A -85,B 0,C 180,E1 4442.221,E2 4442.221} C_VEL
LIN {X 0,Y 291.731,Z 978.898,A -85,B 0,C 180,E1 4441.263,E2 4441.263} C_VEL
LIN {X 0,Y 278.736,Z 999.853,A -85,B 0,C 180,E1 4440.299,E2 4440.299} C_VEL
LIN {X 0,Y 262.182,Z 1023.741,A -85,B 0,C 180,E1 4438.969,E2 4438.969} C_VEL
LIN {X 0,Y 246.357,Z 1044.007,A -85,B 0,C 180,E1 4437.561,E2 4437.561} C_VEL
LIN {X 0,Y 231.118,Z 1061.769,A -85,B 0,C 180,E1 4436.048,E2 4436.048} C_VEL
LIN {X 0,Y 210.828,Z 1083.009,A -85,B 0,C 180,E1 4433.746,E2 4433.746} C_VEL
LIN {X 0,Y 193.858,Z 1098.939,A -85,B 0,C 180,E1 4431.482,E2 4431.482} C_VEL
LIN {X 0,Y 177.591,Z 1112.934,A -85,B 0,C 180,E1 4428.934,E2 4428.934} C_VEL
LIN {X 0,Y 156.994,Z 1129.088,A -85,B 0,C 180,E1 4424.967,E2 4424.967} C_VEL
LIN {X 0,Y 138.549,Z 1142.088,A -85,B 0,C 180,E1 4420.394,E2 4420.394} C_VEL
LIN {X 0,Y 123.106,Z 1152.227,A -85,B 0,C 180,E1 4415.405,E2 4415.405} C_VEL
LIN {X 0,Y 108.01,Z 1161.631,A -85,B 0,C 180,E1 4408.875,E2 4408.875} C_VEL
LIN {X 0,Y 91.011,Z 1171.986,A -85,B 0,C 180,E1 4397.905,E2 4397.905} C_VEL
LIN {X 0,Y 78.687,Z 1179.868,A -85,B 0,C 180,E1 4384.403,E2 4384.403} C_VEL
LIN {X 0,Y 71.738,Z 1185.607,A -85,B 0,C 180,E1 4370.05,E2 4370.05} C_VEL
LIN {X 0,Y 68.898,Z 1190.095,A -85,B 0,C 180,E1 4355.487,E2 4355.487} C_VEL
LIN {X 0,Y 68.869,Z 1193.831,A -85,B 0,C 180,E1 4341.283,E2 4341.283} C_VEL
LIN {X 0,Y 71.992,Z 1197.611,A -85,B 0,C 180,E1 4325.579,E2 4325.579} C_VEL
LIN {X 0,Y 82.545,Z 1201.968,A -85,B 0,C 180,E1 4306.694,E2 4306.694} C_VEL
LIN {X 0,Y 96.171,Z 1204.972,A -85,B 0,C 180,E1 4294.639,E2 4294.639} C_VEL
LIN {X 0,Y 78.677,Z 1209.489,A -85,B 0,C 180,E1 4278.573,E2 4278.573} C_VEL
LIN {X 0,Y 70.215,Z 1212.157,A -85,B 0,C 180,E1 4260.84,E2 4260.84} C_VEL
LIN {X 0,Y 68.356,Z 1213.543,A -85,B 0,C 180,E1 4243.535,E2 4243.535} C_VEL
LIN {X 0,Y 69.654,Z 1213.825,A -85,B 0,C 180,E1 4231.645,E2 4231.645} C_VEL
LIN {X 0,Y 69.713,Z 1213.638,A -85,B 0,C 180,E1 4228.356,E2 4228.356} C_VEL
LIN {X 0,Y 68.704,Z 1211.768,A -85,B 0,C 180,E1 4215.676,E2 4215.676} C_VEL
LIN {X 0,Y 71.694,Z 1207.364,A -85,B 0,C 180,E1 4196.803,E2 4196.803} C_VEL
LIN {X 0,Y 79.9,Z 1201.535,A -85,B 0,C 180,E1 4181.336,E2 4181.336} C_VEL
LIN {X 0,Y 91.19,Z 1194.839,A -85,B 0,C 180,E1 4169.978,E2 4169.978} C_VEL
LIN {X 0,Y 104.294,Z 1187.25,A -85,B 0,C 180,E1 4161.573,E2 4161.573} C_VEL
LIN {X 0,Y 119.054,Z 1178.405,A -85,B 0,C 180,E1 4155.022,E2 4155.022} C_VEL
LIN {X 0,Y 138.647,Z 1165.85,A -85,B 0,C 180,E1 4148.886,E2 4148.886} C_VEL
LIN {X 0,Y 157.488,Z 1152.393,A -85,B 0,C 180,E1 4144.6,E2 4144.6} C_VEL
LIN {X 0,Y 173.066,Z 1140.317,A -85,B 0,C 180,E1 4141.822,E2 4141.822} C_VEL
LIN {X 0,Y 189.714,Z 1126.289,A -85,B 0,C 180,E1 4139.396,E2 4139.396} C_VEL
LIN {X 0,Y 209.909,Z 1107.521,A -85,B 0,C 180,E1 4136.996,E2 4136.996} C_VEL
LIN {X 0,Y 227.487,Z 1089.219,A -85,B 0,C 180,E1 4135.287,E2 4135.287} C_VEL
LIN {X 0,Y 242.791,Z 1071.761,A -85,B 0,C 180,E1 4134.019,E2 4134.019} C_VEL
LIN {X 0,Y 260.895,Z 1048.883,A -85,B 0,C 180,E1 4132.734,E2 4132.734} C_VEL
LIN {X 0,Y 275.766,Z 1027.729,A -85,B 0,C 180,E1 4131.828,E2 4131.828} C_VEL
LIN {X 0,Y 282.446,Z 1017.638,A -85,B 0,C 180,E1 4131.46,E2 4131.46} C_VEL
LIN {X 0,Y 286.106,Z 1011.178,A -85,B 0,C 180,E1 4131.063,E2 4131.063} C_VEL
LIN {X 0,Y 294.102,Z 994.519,A -85,B 0,C 180,E1 4129.482,E2 4129.482} C_VEL
LIN {X 0,Y 297.65,Z 987.734,A -85,B 0,C 180,E1 4129.145,E2 4129.145} C_VEL
LIN {X 0,Y 312.086,Z 959.768,A -85,B 0,C 180,E1 4128.631,E2 4128.631} C_VEL
LIN {X 0,Y 322.647,Z 936.306,A -85,B 0,C 180,E1 4128.315,E2 4128.315} C_VEL
LIN {X 0,Y 333.471,Z 908.575,A -85,B 0,C 180,E1 4128.021,E2 4128.021} C_VEL
LIN {X 0,Y 341.924,Z 882.038,A -85,B 0,C 180,E1 4127.726,E2 4127.726} C_VEL
LIN {X 0,Y 348.767,Z 856.06,A -85,B 0,C 180,E1 4127.429,E2 4127.429} C_VEL
LIN {X 0,Y 356.554,Z 817.417,A -85,B 0,C 180,E1 4127.024,E2 4127.024} C_VEL
LIN {X 0,Y 368.893,Z 751.01,A -85,B 0,C 180,E1 4126.36,E2 4126.36} C_VEL
LIN {X 0,Y 365.608,Z 744.852,A -85,B 0,C 180,E1 4122.328,E2 4122.328} C_VEL
LIN {X 0,Y 363.993,Z 741.672,A -85,B 0,C 180,E1 4119.917,E2 4119.917} C_VEL
LIN {X 0,Y 363.055,Z 740.286,A -85,B 0,C 180,E1 4118.343,E2 4118.343} C_VEL
LIN {X 0,Y 360.474,Z 736.622,A -85,B 0,C 180,E1 4112.922,E2 4112.922} C_VEL
LIN {X 0,Y 360.091,Z 735.509,A -85,B 0,C 180,E1 4111.289,E2 4111.289} C_VEL
LIN {X 0,Y 359.046,Z 734.902,A -85,B 0,C 180,E1 4105.801,E2 4105.801} C_VEL
LIN {X 0,Y 359.441,Z 735.017,A -85,B 0,C 180,E1 4101.047,E2 4101.047} C_VEL
LIN {X 0,Y 360.856,Z 735.834,A -85,B 0,C 180,E1 4096.549,E2 4096.549} C_VEL
LIN {X 0,Y 363.658,Z 740.065,A -85,B 0,C 180,E1 4090.873,E2 4090.873} C_VEL
LIN {X 0,Y 364.796,Z 741.438,A -85,B 0,C 180,E1 4089.283,E2 4089.283} C_VEL
LIN {X 0,Y 366.404,Z 743.992,A -85,B 0,C 180,E1 4087.147,E2 4087.147} C_VEL
LIN {X 0,Y 351.877,Z 820.643,A -85,B 0,C 180,E1 4086.4,E2 4086.4} C_VEL
LIN {X 0,Y 344.404,Z 850.739,A -85,B 0,C 180,E1 4085.997,E2 4085.997} C_VEL
LIN {X 0,Y 336.776,Z 875.845,A -85,B 0,C 180,E1 4085.585,E2 4085.585} C_VEL
LIN {X 0,Y 325.833,Z 905.908,A -85,B 0,C 180,E1 4084.98,E2 4084.98} C_VEL
LIN {X 0,Y 315.858,Z 929.265,A -85,B 0,C 180,E1 4084.406,E2 4084.406} C_VEL
LIN {X 0,Y 303.193,Z 955.415,A -85,B 0,C 180,E1 4083.644,E2 4083.644} C_VEL
LIN {X 0,Y 289.39,Z 979.975,A -85,B 0,C 180,E1 4082.764,E2 4082.764} C_VEL
LIN {X 0,Y 276.446,Z 1000.661,A -85,B 0,C 180,E1 4081.875,E2 4081.875} C_VEL
LIN {X 0,Y 259.901,Z 1024.363,A -85,B 0,C 180,E1 4080.647,E2 4080.647} C_VEL
LIN {X 0,Y 243.897,Z 1044.665,A -85,B 0,C 180,E1 4079.334,E2 4079.334} C_VEL
LIN {X 0,Y 228.624,Z 1062.291,A -85,B 0,C 180,E1 4077.938,E2 4077.938} C_VEL
LIN {X 0,Y 208.956,Z 1082.782,A -85,B 0,C 180,E1 4075.892,E2 4075.892} C_VEL
LIN {X 0,Y 191.125,Z 1099.341,A -85,B 0,C 180,E1 4073.718,E2 4073.718} C_VEL
LIN {X 0,Y 175.075,Z 1112.99,A -85,B 0,C 180,E1 4071.419,E2 4071.419} C_VEL
LIN {X 0,Y 156.621,Z 1127.381,A -85,B 0,C 180,E1 4068.229,E2 4068.229} C_VEL
LIN {X 0,Y 135.799,Z 1141.955,A -85,B 0,C 180,E1 4063.608,E2 4063.608} C_VEL
LIN {X 0,Y 119.101,Z 1152.661,A -85,B 0,C 180,E1 4058.692,E2 4058.692} C_VEL
LIN {X 0,Y 103.641,Z 1161.94,A -85,B 0,C 180,E1 4052.545,E2 4052.545} C_VEL
LIN {X 0,Y 86.853,Z 1171.65,A -85,B 0,C 180,E1 4042.725,E2 4042.725} C_VEL
LIN {X 0,Y 71.603,Z 1180.738,A -85,B 0,C 180,E1 4027.169,E2 4027.169} C_VEL
LIN {X 0,Y 63.881,Z 1186.679,A -85,B 0,C 180,E1 4011.239,E2 4011.239} C_VEL
LIN {X 0,Y 60.862,Z 1191.237,A -85,B 0,C 180,E1 3994.773,E2 3994.773} C_VEL
LIN {X 0,Y 61.156,Z 1195.14,A -85,B 0,C 180,E1 3978.509,E2 3978.509} C_VEL
LIN {X 0,Y 65.719,Z 1199.255,A -85,B 0,C 180,E1 3960,E2 3960} C_VEL
LIN {X 0,Y 79.196,Z 1203.863,A -85,B 0,C 180,E1 3940.069,E2 3940.069} C_VEL
LIN {X 0,Y 85.459,Z 1205.269,A -85,B 0,C 180,E1 3934.719,E2 3934.719} C_VEL
LIN {X 0,Y 67.658,Z 1209.328,A -85,B 0,C 180,E1 3915.182,E2 3915.182} C_VEL
LIN {X 0,Y 60.746,Z 1211.517,A -85,B 0,C 180,E1 3892.245,E2 3892.245} C_VEL
LIN {X 0,Y 61.318,Z 1212.129,A -85,B 0,C 180,E1 3874.676,E2 3874.676} C_VEL
LIN {X 0,Y 61.995,Z 1211.999,A -85,B 0,C 180,E1 3869.556,E2 3869.556} C_VEL
LIN {X 0,Y 60.854,Z 1210.22,A -85,B 0,C 180,E1 3855.732,E2 3855.732} C_VEL
LIN {X 0,Y 64.196,Z 1205.77,A -85,B 0,C 180,E1 3834.81,E2 3834.81} C_VEL
LIN {X 0,Y 72.916,Z 1200.173,A -85,B 0,C 180,E1 3818.59,E2 3818.59} C_VEL
LIN {X 0,Y 84.366,Z 1193.898,A -85,B 0,C 180,E1 3807.267,E2 3807.267} C_VEL
LIN {X 0,Y 98.16,Z 1186.399,A -85,B 0,C 180,E1 3798.681,E2 3798.681} C_VEL
LIN {X 0,Y 113.54,Z 1177.638,A -85,B 0,C 180,E1 3792.175,E2 3792.175} C_VEL
LIN {X 0,Y 132.827,Z 1165.813,A -85,B 0,C 180,E1 3786.46,E2 3786.46} C_VEL
LIN {X 0,Y 153.088,Z 1151.859,A -85,B 0,C 180,E1 3782.138,E2 3782.138} C_VEL
LIN {X 0,Y 170.287,Z 1138.826,A -85,B 0,C 180,E1 3779.327,E2 3779.327} C_VEL
LIN {X 0,Y 188.332,Z 1123.834,A -85,B 0,C 180,E1 3776.957,E2 3776.957} C_VEL
LIN {X 0,Y 209.306,Z 1104.362,A -85,B 0,C 180,E1 3774.74,E2 3774.74} C_VEL
LIN {X 0,Y 225.499,Z 1087.638,A -85,B 0,C 180,E1 3773.329,E2 3773.329} C_VEL
LIN {X 0,Y 241.41,Z 1069.621,A -85,B 0,C 180,E1 3772.144,E2 3772.144} C_VEL
LIN {X 0,Y 260.398,Z 1045.564,A -85,B 0,C 180,E1 3770.942,E2 3770.942} C_VEL
LIN {X 0,Y 274.621,Z 1025.378,A -85,B 0,C 180,E1 3770.176,E2 3770.176} C_VEL
LIN {X 0,Y 289.85,Z 1001.429,A -85,B 0,C 180,E1 3769.465,E2 3769.465} C_VEL
LIN {X 0,Y 297.65,Z 987.734,A -85,B 0,C 180,E1 3769.145,E2 3769.145} C_VEL
LIN {X 0,Y 301.101,Z 980.999,A -85,B 0,C 180,E1 3768.822,E2 3768.822} C_VEL
LIN {X 0,Y 308.74,Z 962.821,A -85,B 0,C 180,E1 3767.382,E2 3767.382} C_VEL
LIN {X 0,Y 311.415,Z 956.707,A -85,B 0,C 180,E1 3767.168,E2 3767.168} C_VEL
LIN {X 0,Y 322.356,Z 932.325,A -85,B 0,C 180,E1 3766.895,E2 3766.895} C_VEL
LIN {X 0,Y 333.171,Z 903.924,A -85,B 0,C 180,E1 3766.639,E2 3766.639} C_VEL
LIN {X 0,Y 340.977,Z 879.197,A -85,B 0,C 180,E1 3766.385,E2 3766.385} C_VEL
LIN {X 0,Y 348.461,Z 850.291,A -85,B 0,C 180,E1 3766.078,E2 3766.078} C_VEL
LIN {X 0,Y 359.572,Z 793.096,A -85,B 0,C 180,E1 3765.535,E2 3765.535} C_VEL
LIN {X 0,Y 366.298,Z 757.209,A -85,B 0,C 180,E1 3765.179,E2 3765.179} C_VEL
LIN {X 0,Y 363.538,Z 751.768,A -85,B 0,C 180,E1 3761.561,E2 3761.561} C_VEL
LIN {X 0,Y 361.742,Z 748.353,A -85,B 0,C 180,E1 3758.771,E2 3758.771} C_VEL
LIN {X 0,Y 358.927,Z 744.615,A -85,B 0,C 180,E1 3753.054,E2 3753.054} C_VEL
LIN {X 0,Y 358.479,Z 743.331,A -85,B 0,C 180,E1 3751.141,E2 3751.141} C_VEL
LIN {X 0,Y 357.472,Z 742.746,A -85,B 0,C 180,E1 3745.79,E2 3745.79} C_VEL
LIN {X 0,Y 357.871,Z 742.862,A -85,B 0,C 180,E1 3741.049,E2 3741.049} C_VEL
LIN {X 0,Y 359.279,Z 743.724,A -85,B 0,C 180,E1 3736.574,E2 3736.574} C_VEL
LIN {X 0,Y 362.135,Z 747.958,A -85,B 0,C 180,E1 3730.839,E2 3730.839} C_VEL
LIN {X 0,Y 363.275,Z 749.462,A -85,B 0,C 180,E1 3729.224,E2 3729.224} C_VEL
LIN {X 0,Y 363.879,Z 750.695,A -85,B 0,C 180,E1 3728.327,E2 3728.327} C_VEL
LIN {X 0,Y 350.142,Z 822.237,A -85,B 0,C 180,E1 3727.669,E2 3727.669} C_VEL
LIN {X 0,Y 342.676,Z 851.914,A -85,B 0,C 180,E1 3727.294,E2 3727.294} C_VEL
LIN {X 0,Y 335.032,Z 876.842,A -85,B 0,C 180,E1 3726.912,E2 3726.912} C_VEL
LIN {X 0,Y 323.936,Z 907.065,A -85,B 0,C 180,E1 3726.344,E2 3726.344} C_VEL
LIN {X 0,Y 313.577,Z 931.078,A -85,B 0,C 180,E1 3725.792,E2 3725.792} C_VEL
LIN {X 0,Y 300.535,Z 957.6,A -85,B 0,C 180,E1 3725.07,E2 3725.07} C_VEL
LIN {X 0,Y 286.712,Z 981.897,A -85,B 0,C 180,E1 3724.256,E2 3724.256} C_VEL
LIN {X 0,Y 273.045,Z 1003.452,A -85,B 0,C 180,E1 3723.39,E2 3723.39} C_VEL
LIN {X 0,Y 255.134,Z 1028.444,A -85,B 0,C 180,E1 3722.164,E2 3722.164} C_VEL
LIN {X 0,Y 240.411,Z 1046.821,A -85,B 0,C 180,E1 3721.043,E2 3721.043} C_VEL
LIN {X 0,Y 223.568,Z 1065.93,A -85,B 0,C 180,E1 3719.618,E2 3719.618} C_VEL
LIN {X 0,Y 204.081,Z 1085.646,A -85,B 0,C 180,E1 3717.739,E2 3717.739} C_VEL
LIN {X 0,Y 187.039,Z 1101.197,A -85,B 0,C 180,E1 3715.818,E2 3715.818} C_VEL
LIN {X 0,Y 169.391,Z 1115.888,A -85,B 0,C 180,E1 3713.471,E2 3713.471} C_VEL
LIN {X 0,Y 146.535,Z 1132.894,A -85,B 0,C 180,E1 3709.668,E2 3709.668} C_VEL
LIN {X 0,Y 128.588,Z 1144.869,A -85,B 0,C 180,E1 3705.793,E2 3705.793} C_VEL
LIN {X 0,Y 112.089,Z 1155.014,A -85,B 0,C 180,E1 3701.11,E2 3701.11} C_VEL
LIN {X 0,Y 93.168,Z 1165.895,A -85,B 0,C 180,E1 3693.534,E2 3693.534} C_VEL
LIN {X 0,Y 74.708,Z 1175.898,A -85,B 0,C 180,E1 3681.534,E2 3681.534} C_VEL
LIN {X 0,Y 62.724,Z 1182.795,A -85,B 0,C 180,E1 3667.507,E2 3667.507} C_VEL
LIN {X 0,Y 55.167,Z 1188.523,A -85,B 0,C 180,E1 3649.574,E2 3649.574} C_VEL
LIN {X 0,Y 52.728,Z 1192.757,A -85,B 0,C 180,E1 3632.071,E2 3632.071} C_VEL
LIN {X 0,Y 53.743,Z 1196.591,A -85,B 0,C 180,E1 3613.997,E2 3613.997} C_VEL
LIN {X 0,Y 61.031,Z 1201.25,A -85,B 0,C 180,E1 3591.521,E2 3591.521} C_VEL
LIN {X 0,Y 74.675,Z 1205.258,A -85,B 0,C 180,E1 3574.83,E2 3574.83} C_VEL
LIN {X 0,Y 56.558,Z 1208.911,A -85,B 0,C 180,E1 3549.526,E2 3549.526} C_VEL
LIN {X 0,Y 52.706,Z 1210.232,A -85,B 0,C 180,E1 3523.158,E2 3523.158} C_VEL
LIN {X 0,Y 54.155,Z 1210.207,A -85,B 0,C 180,E1 3510,E2 3510} C_VEL
LIN {X 0,Y 53.046,Z 1208.325,A -85,B 0,C 180,E1 3494.011,E2 3494.011} C_VEL
LIN {X 0,Y 56.886,Z 1204.12,A -85,B 0,C 180,E1 3472.034,E2 3472.034} C_VEL
LIN {X 0,Y 66.451,Z 1198.625,A -85,B 0,C 180,E1 3454.875,E2 3454.875} C_VEL
LIN {X 0,Y 78.524,Z 1192.523,A -85,B 0,C 180,E1 3443.536,E2 3443.536} C_VEL
LIN {X 0,Y 93.45,Z 1184.877,A -85,B 0,C 180,E1 3434.88,E2 3434.88} C_VEL
LIN {X 0,Y 109.26,Z 1176.265,A -85,B 0,C 180,E1 3428.755,E2 3428.755} C_VEL
LIN {X 0,Y 129.208,Z 1164.442,A -85,B 0,C 180,E1 3423.375,E2 3423.375} C_VEL
LIN {X 0,Y 149.99,Z 1150.453,A -85,B 0,C 180,E1 3419.375,E2 3419.375} C_VEL
LIN {X 0,Y 167.234,Z 1137.65,A -85,B 0,C 180,E1 3416.839,E2 3416.839} C_VEL
LIN {X 0,Y 183.712,Z 1124.243,A -85,B 0,C 180,E1 3414.873,E2 3414.873} C_VEL
LIN {X 0,Y 204.042,Z 1105.974,A -85,B 0,C 180,E1 3412.894,E2 3412.894} C_VEL
LIN {X 0,Y 222.453,Z 1087.31,A -85,B 0,C 180,E1 3411.437,E2 3411.437} C_VEL
LIN {X 0,Y 237.93,Z 1070.053,A -85,B 0,C 180,E1 3410.399,E2 3410.399} C_VEL
LIN {X 0,Y 256.39,Z 1047.22,A -85,B 0,C 180,E1 3409.344,E2 3409.344} C_VEL
LIN {X 0,Y 271.667,Z 1025.878,A -85,B 0,C 180,E1 3408.603,E2 3408.603} C_VEL
LIN {X 0,Y 285.691,Z 1004.186,A -85,B 0,C 180,E1 3408.017,E2 3408.017} C_VEL
LIN {X 0,Y 301.132,Z 977.113,A -85,B 0,C 180,E1 3407.473,E2 3407.473} C_VEL
LIN {X 0,Y 311.415,Z 956.707,A -85,B 0,C 180,E1 3407.168,E2 3407.168} C_VEL
LIN {X 0,Y 314.456,Z 949.759,A -85,B 0,C 180,E1 3406.905,E2 3406.905} C_VEL
LIN {X 0,Y 321.233,Z 930.855,A -85,B 0,C 180,E1 3405.626,E2 3405.626} C_VEL
LIN {X 0,Y 323.523,Z 924.679,A -85,B 0,C 180,E1 3405.453,E2 3405.453} C_VEL
LIN {X 0,Y 332.653,Z 899.963,A -85,B 0,C 180,E1 3405.263,E2 3405.263} C_VEL
LIN {X 0,Y 340.373,Z 875.238,A -85,B 0,C 180,E1 3405.032,E2 3405.032} C_VEL
LIN {X 0,Y 348.122,Z 844.142,A -85,B 0,C 180,E1 3404.731,E2 3404.731} C_VEL
LIN {X 0,Y 363.672,Z 763.339,A -85,B 0,C 180,E1 3404,E2 3404} C_VEL
LIN {X 0,Y 360.799,Z 757.514,A -85,B 0,C 180,E1 3399.901,E2 3399.901} C_VEL
LIN {X 0,Y 359.793,Z 755.899,A -85,B 0,C 180,E1 3398.136,E2 3398.136} C_VEL
LIN {X 0,Y 357.225,Z 752.214,A -85,B 0,C 180,E1 3392.674,E2 3392.674} C_VEL
LIN {X 0,Y 356.859,Z 751.147,A -85,B 0,C 180,E1 3390.949,E2 3390.949} C_VEL
LIN {X 0,Y 355.891,Z 750.582,A -85,B 0,C 180,E1 3385.617,E2 3385.617} C_VEL
LIN {X 0,Y 356.406,Z 750.759,A -85,B 0,C 180,E1 3380.651,E2 3380.651} C_VEL
LIN {X 0,Y 357.698,Z 751.598,A -85,B 0,C 180,E1 3376.617,E2 3376.617} C_VEL
LIN {X 0,Y 360.56,Z 755.805,A -85,B 0,C 180,E1 3370.878,E2 3370.878} C_VEL
LIN {X 0,Y 361.522,Z 757.072,A -85,B 0,C 180,E1 3369.524,E2 3369.524} C_VEL
LIN {X 0,Y 348.749,Z 823.018,A -85,B 0,C 180,E1 3368.958,E2 3368.958} C_VEL
LIN {X 0,Y 341.218,Z 852.734,A -85,B 0,C 180,E1 3368.608,E2 3368.608} C_VEL
LIN {X 0,Y 333.635,Z 877.306,A -85,B 0,C 180,E1 3368.26,E2 3368.26} C_VEL
LIN {X 0,Y 322.687,Z 907.065,A -85,B 0,C 180,E1 3367.746,E2 3367.746} C_VEL
LIN {X 0,Y 312.281,Z 931.105,A -85,B 0,C 180,E1 3367.24,E2 3367.24} C_VEL
LIN {X 0,Y 299.314,Z 957.468,A -85,B 0,C 180,E1 3366.584,E2 3366.584} C_VEL
LIN {X 0,Y 284.811,Z 982.813,A -85,B 0,C 180,E1 3365.808,E2 3365.808} C_VEL
LIN {X 0,Y 271.034,Z 1004.367,A -85,B 0,C 180,E1 3365.015,E2 3365.015} C_VEL
LIN {X 0,Y 252.858,Z 1029.516,A -85,B 0,C 180,E1 3363.887,E2 3363.887} C_VEL
LIN {X 0,Y 237.793,Z 1048.123,A -85,B 0,C 180,E1 3362.849,E2 3362.849} C_VEL
LIN {X 0,Y 219.616,Z 1068.47,A -85,B 0,C 180,E1 3361.453,E2 3361.453} C_VEL
LIN {X 0,Y 199.755,Z 1088.094,A -85,B 0,C 180,E1 3359.706,E2 3359.706} C_VEL
LIN {X 0,Y 183.147,Z 1102.959,A -85,B 0,C 180,E1 3358.003,E2 3358.003} C_VEL
LIN {X 0,Y 165.196,Z 1117.615,A -85,B 0,C 180,E1 3355.836,E2 3355.836} C_VEL
LIN {X 0,Y 142.83,Z 1133.93,A -85,B 0,C 180,E1 3352.47,E2 3352.47} C_VEL
LIN {X 0,Y 124.753,Z 1145.753,A -85,B 0,C 180,E1 3348.956,E2 3348.956} C_VEL
LIN {X 0,Y 107.409,Z 1156.156,A -85,B 0,C 180,E1 3344.496,E2 3344.496} C_VEL
LIN {X 0,Y 87.611,Z 1167.091,A -85,B 0,C 180,E1 3337.212,E2 3337.212} C_VEL
LIN {X 0,Y 68.219,Z 1177.019,A -85,B 0,C 180,E1 3325.335,E2 3325.335} C_VEL
LIN {X 0,Y 54.788,Z 1184.226,A -85,B 0,C 180,E1 3309.712,E2 3309.712} C_VEL
LIN {X 0,Y 47.003,Z 1189.786,A -85,B 0,C 180,E1 3289.982,E2 3289.982} C_VEL
LIN {X 0,Y 44.703,Z 1193.76,A -85,B 0,C 180,E1 3270.961,E2 3270.961} C_VEL
LIN {X 0,Y 46.304,Z 1197.722,A -85,B 0,C 180,E1 3249.948,E2 3249.948} C_VEL
LIN {X 0,Y 56.622,Z 1202.879,A -85,B 0,C 180,E1 3223.588,E2 3223.588} C_VEL
LIN {X 0,Y 63.749,Z 1204.92,A -85,B 0,C 180,E1 3214.802,E2 3214.802} C_VEL
LIN {X 0,Y 48.708,Z 1207.426,A -85,B 0,C 180,E1 3191.063,E2 3191.063} C_VEL
LIN {X 0,Y 44.949,Z 1208.471,A -85,B 0,C 180,E1 3161.823,E2 3161.823} C_VEL
LIN {X 0,Y 46.237,Z 1208.396,A -85,B 0,C 180,E1 3150,E2 3150} C_VEL
LIN {X 0,Y 45.28,Z 1206.367,A -85,B 0,C 180,E1 3131.723,E2 3131.723} C_VEL
LIN {X 0,Y 49.756,Z 1202.398,A -85,B 0,C 180,E1 3108.459,E2 3108.459} C_VEL
LIN {X 0,Y 59.632,Z 1197.361,A -85,B 0,C 180,E1 3091.225,E2 3091.225} C_VEL
LIN {X 0,Y 73.213,Z 1191.049,A -85,B 0,C 180,E1 3079.134,E2 3079.134} C_VEL
LIN {X 0,Y 88.602,Z 1183.64,A -85,B 0,C 180,E1 3070.947,E2 3070.947} C_VEL
LIN {X 0,Y 106.36,Z 1174.388,A -85,B 0,C 180,E1 3064.797,E2 3064.797} C_VEL
LIN {X 0,Y 128.988,Z 1161.137,A -85,B 0,C 180,E1 3059.538,E2 3059.538} C_VEL
LIN {X 0,Y 148.281,Z 1148.337,A -85,B 0,C 180,E1 3056.357,E2 3056.357} C_VEL
LIN {X 0,Y 165.856,Z 1135.447,A -85,B 0,C 180,E1 3054.109,E2 3054.109} C_VEL
LIN {X 0,Y 186.801,Z 1118.422,A -85,B 0,C 180,E1 3051.986,E2 3051.986} C_VEL
LIN {X 0,Y 206.36,Z 1100.352,A -85,B 0,C 180,E1 3050.408,E2 3050.408} C_VEL
LIN {X 0,Y 222.85,Z 1083.547,A -85,B 0,C 180,E1 3049.296,E2 3049.296} C_VEL
LIN {X 0,Y 241.544,Z 1062.449,A -85,B 0,C 180,E1 3048.236,E2 3048.236} C_VEL
LIN {X 0,Y 258.144,Z 1041.242,A -85,B 0,C 180,E1 3047.443,E2 3047.443} C_VEL
LIN {X 0,Y 272.616,Z 1020.817,A -85,B 0,C 180,E1 3046.856,E2 3046.856} C_VEL
LIN {X 0,Y 289.213,Z 994.417,A -85,B 0,C 180,E1 3046.284,E2 3046.284} C_VEL
LIN {X 0,Y 301.506,Z 972.22,A -85,B 0,C 180,E1 3045.932,E2 3045.932} C_VEL
LIN {X 0,Y 314.249,Z 946.371,A -85,B 0,C 180,E1 3045.63,E2 3045.63} C_VEL
LIN {X 0,Y 323.523,Z 924.679,A -85,B 0,C 180,E1 3045.453,E2 3045.453} C_VEL
LIN {X 0,Y 326.146,Z 917.447,A -85,B 0,C 180,E1 3045.25,E2 3045.25} C_VEL
LIN {X 0,Y 329.545,Z 906.309,A -85,B 0,C 180,E1 3044.555,E2 3044.555} C_VEL
LIN {X 0,Y 332.374,Z 896.056,A -85,B 0,C 180,E1 3043.949,E2 3043.949} C_VEL
LIN {X 0,Y 333.705,Z 891.851,A -85,B 0,C 180,E1 3043.848,E2 3043.848} C_VEL
LIN {X 0,Y 342.281,Z 862.264,A -85,B 0,C 180,E1 3043.597,E2 3043.597} C_VEL
LIN {X 0,Y 348.156,Z 836.912,A -85,B 0,C 180,E1 3043.373,E2 3043.373} C_VEL
LIN {X 0,Y 361.169,Z 769.424,A -85,B 0,C 180,E1 3042.81,E2 3042.81} C_VEL
LIN {X 0,Y 358.834,Z 764.762,A -85,B 0,C 180,E1 3039.275,E2 3039.275} C_VEL
LIN {X 0,Y 357.886,Z 763.483,A -85,B 0,C 180,E1 3037.632,E2 3037.632} C_VEL
LIN {X 0,Y 355.514,Z 759.71,A -85,B 0,C 180,E1 3032.168,E2 3032.168} C_VEL
LIN {X 0,Y 355.181,Z 758.942,A -85,B 0,C 180,E1 3030.67,E2 3030.67} C_VEL
LIN {X 0,Y 354.313,Z 758.419,A -85,B 0,C 180,E1 3025.442,E2 3025.442} C_VEL
LIN {X 0,Y 354.953,Z 758.657,A -85,B 0,C 180,E1 3020.249,E2 3020.249} C_VEL
LIN {X 0,Y 356.12,Z 759.478,A -85,B 0,C 180,E1 3016.651,E2 3016.651} C_VEL
LIN {X 0,Y 359.011,Z 763.675,A -85,B 0,C 180,E1 3010.881,E2 3010.881} C_VEL
LIN {X 0,Y 359.071,Z 764.02,A -85,B 0,C 180,E1 3010.729,E2 3010.729} C_VEL
LIN {X 0,Y 346.924,Z 825.719,A -85,B 0,C 180,E1 3010.235,E2 3010.235} C_VEL
LIN {X 0,Y 339.336,Z 854.94,A -85,B 0,C 180,E1 3009.912,E2 3009.912} C_VEL
LIN {X 0,Y 330.917,Z 881.72,A -85,B 0,C 180,E1 3009.558,E2 3009.558} C_VEL
LIN {X 0,Y 319.934,Z 910.672,A -85,B 0,C 180,E1 3009.088,E2 3009.088} C_VEL
LIN {X 0,Y 309.768,Z 933.794,A -85,B 0,C 180,E1 3008.634,E2 3008.634} C_VEL
LIN {X 0,Y 296.146,Z 960.884,A -85,B 0,C 180,E1 3008.012,E2 3008.012} C_VEL
LIN {X 0,Y 282.611,Z 984.275,A -85,B 0,C 180,E1 3007.356,E2 3007.356} C_VEL
LIN {X 0,Y 268.244,Z 1006.539,A -85,B 0,C 180,E1 3006.612,E2 3006.612} C_VEL
LIN {X 0,Y 250.599,Z 1030.668,A -85,B 0,C 180,E1 3005.629,E2 3005.629} C_VEL
LIN {X 0,Y 235.399,Z 1049.287,A -85,B 0,C 180,E1 3004.693,E2 3004.693} C_VEL
LIN {X 0,Y 217.543,Z 1069.119,A -85,B 0,C 180,E1 3003.473,E2 3003.473} C_VEL
LIN {X 0,Y 197.606,Z 1088.696,A -85,B 0,C 180,E1 3001.922,E2 3001.922} C_VEL
LIN {X 0,Y 180.866,Z 1103.567,A -85,B 0,C 180,E1 3000.41,E2 3000.41} C_VEL
LIN {X 0,Y 162.672,Z 1118.274,A -85,B 0,C 180,E1 2998.481,E2 2998.481} C_VEL
LIN {X 0,Y 139.067,Z 1135.254,A -85,B 0,C 180,E1 2995.351,E2 2995.351} C_VEL
LIN {X 0,Y 120.994,Z 1146.801,A -85,B 0,C 180,E1 2992.246,E2 2992.246} C_VEL
LIN {X 0,Y 103.14,Z 1157.194,A -85,B 0,C 180,E1 2988.183,E2 2988.183} C_VEL
LIN {X 0,Y 83.796,Z 1167.506,A -85,B 0,C 180,E1 2981.913,E2 2981.913} C_VEL
LIN {X 0,Y 61.994,Z 1178.18,A -85,B 0,C 180,E1 2969.833,E2 2969.833} C_VEL
LIN {X 0,Y 47.821,Z 1185.167,A -85,B 0,C 180,E1 2954.119,E2 2954.119} C_VEL
LIN {X 0,Y 39.176,Z 1190.668,A -85,B 0,C 180,E1 2932.227,E2 2932.227} C_VEL
LIN {X 0,Y 36.695,Z 1194.771,A -85,B 0,C 180,E1 2909.317,E2 2909.317} C_VEL
LIN {X 0,Y 39.141,Z 1198.708,A -85,B 0,C 180,E1 2884.396,E2 2884.396} C_VEL
LIN {X 0,Y 52.924,Z 1204.359,A -85,B 0,C 180,E1 2855.071,E2 2855.071} C_VEL
LIN {X 0,Y 38.606,Z 1206.275,A -85,B 0,C 180,E1 2824.026,E2 2824.026} C_VEL
LIN {X 0,Y 37.741,Z 1206.571,A -85,B 0,C 180,E1 2794.558,E2 2794.558} C_VEL
LIN {X 0,Y 38.312,Z 1206.537,A -85,B 0,C 180,E1 2789.999,E2 2789.999} C_VEL
LIN {X 0,Y 37.733,Z 1204.176,A -85,B 0,C 180,E1 2766.579,E2 2766.579} C_VEL
LIN {X 0,Y 43.378,Z 1200.445,A -85,B 0,C 180,E1 2742.471,E2 2742.471} C_VEL
LIN {X 0,Y 54.76,Z 1195.366,A -85,B 0,C 180,E1 2724.832,E2 2724.832} C_VEL
LIN {X 0,Y 68.968,Z 1189.276,A -85,B 0,C 180,E1 2713.749,E2 2713.749} C_VEL
LIN {X 0,Y 85.763,Z 1181.591,A -85,B 0,C 180,E1 2706.023,E2 2706.023} C_VEL
LIN {X 0,Y 106.987,Z 1170.853,A -85,B 0,C 180,E1 2699.936,E2 2699.936} C_VEL
LIN {X 0,Y 128.317,Z 1158.344,A -85,B 0,C 180,E1 2695.873,E2 2695.873} C_VEL
LIN {X 0,Y 146.526,Z 1146.44,A -85,B 0,C 180,E1 2693.338,E2 2693.338} C_VEL
LIN {X 0,Y 165.301,Z 1132.821,A -85,B 0,C 180,E1 2691.302,E2 2691.302} C_VEL
LIN {X 0,Y 188.208,Z 1114.045,A -85,B 0,C 180,E1 2689.368,E2 2689.368} C_VEL
LIN {X 0,Y 205.382,Z 1098.228,A -85,B 0,C 180,E1 2688.201,E2 2688.201} C_VEL
LIN {X 0,Y 222.481,Z 1080.874,A -85,B 0,C 180,E1 2687.224,E2 2687.224} C_VEL
LIN {X 0,Y 242.388,Z 1058.195,A -85,B 0,C 180,E1 2686.279,E2 2686.279} C_VEL
LIN {X 0,Y 257.369,Z 1039.052,A -85,B 0,C 180,E1 2685.675,E2 2685.675} C_VEL
LIN {X 0,Y 273.097,Z 1016.808,A -85,B 0,C 180,E1 2685.143,E2 2685.143} C_VEL
LIN {X 0,Y 288.637,Z 991.809,A -85,B 0,C 180,E1 2684.706,E2 2684.706} C_VEL
LIN {X 0,Y 301.024,Z 969.381,A -85,B 0,C 180,E1 2684.42,E2 2684.42} C_VEL
LIN {X 0,Y 314.133,Z 942.437,A -85,B 0,C 180,E1 2684.176,E2 2684.176} C_VEL
LIN {X 0,Y 324.751,Z 916.928,A -85,B 0,C 180,E1 2684.026,E2 2684.026} C_VEL
LIN {X 0,Y 333.399,Z 892.754,A -85,B 0,C 180,E1 2683.856,E2 2683.856} C_VEL
LIN {X 0,Y 333.705,Z 891.851,A -85,B 0,C 180,E1 2683.848,E2 2683.848} C_VEL
LIN {X 0,Y 335.896,Z 884.525,A -85,B 0,C 180,E1 2683.621,E2 2683.621} C_VEL
LIN {X 0,Y 340.362,Z 864.96,A -85,B 0,C 180,E1 2682.431,E2 2682.431} C_VEL
LIN {X 0,Y 341.846,Z 858.549,A -85,B 0,C 180,E1 2682.246,E2 2682.246} C_VEL
LIN {X 0,Y 348.321,Z 830.026,A -85,B 0,C 180,E1 2682.017,E2 2682.017} C_VEL
LIN {X 0,Y 358.785,Z 775.808,A -85,B 0,C 180,E1 2681.602,E2 2681.602} C_VEL
LIN {X 0,Y 357.002,Z 772.199,A -85,B 0,C 180,E1 2678.82,E2 2678.82} C_VEL
LIN {X 0,Y 354.138,Z 768.213,A -85,B 0,C 180,E1 2672.962,E2 2672.962} C_VEL
LIN {X 0,Y 353.681,Z 766.823,A -85,B 0,C 180,E1 2670.875,E2 2670.875} C_VEL
LIN {X 0,Y 352.739,Z 766.264,A -85,B 0,C 180,E1 2665.463,E2 2665.463} C_VEL
LIN {X 0,Y 353.386,Z 766.502,A -85,B 0,C 180,E1 2660.248,E2 2660.248} C_VEL
LIN {X 0,Y 354.522,Z 767.314,A -85,B 0,C 180,E1 2656.736,E2 2656.736} C_VEL
LIN {X 0,Y 356.686,Z 771.08,A -85,B 0,C 180,E1 2651.948,E2 2651.948} C_VEL
LIN {X 0,Y 345.459,Z 827.491,A -85,B 0,C 180,E1 2651.53,E2 2651.53} C_VEL
LIN {X 0,Y 337.807,Z 856.528,A -85,B 0,C 180,E1 2651.237,E2 2651.237} C_VEL
LIN {X 0,Y 329.497,Z 882.744,A -85,B 0,C 180,E1 2650.92,E2 2650.92} C_VEL
LIN {X 0,Y 318.672,Z 911.15,A -85,B 0,C 180,E1 2650.503,E2 2650.503} C_VEL
LIN {X 0,Y 308.047,Z 935.179,A -85,B 0,C 180,E1 2650.077,E2 2650.077} C_VEL
LIN {X 0,Y 293.943,Z 962.912,A -85,B 0,C 180,E1 2649.502,E2 2649.502} C_VEL
LIN {X 0,Y 280.659,Z 985.684,A -85,B 0,C 180,E1 2648.929,E2 2648.929} C_VEL
LIN {X 0,Y 265.713,Z 1008.647,A -85,B 0,C 180,E1 2648.244,E2 2648.244} C_VEL
LIN {X 0,Y 248.575,Z 1031.83,A -85,B 0,C 180,E1 2647.401,E2 2647.401} C_VEL
LIN {X 0,Y 233.254,Z 1050.464,A -85,B 0,C 180,E1 2646.573,E2 2646.573} C_VEL
LIN {X 0,Y 214.87,Z 1070.704,A -85,B 0,C 180,E1 2645.476,E2 2645.476} C_VEL
LIN {X 0,Y 194.457,Z 1090.457,A -85,B 0,C 180,E1 2644.088,E2 2644.088} C_VEL
LIN {X 0,Y 177.087,Z 1105.628,A -85,B 0,C 180,E1 2642.722,E2 2642.722} C_VEL
LIN {X 0,Y 155.87,Z 1122.402,A -85,B 0,C 180,E1 2640.728,E2 2640.728} C_VEL
LIN {X 0,Y 133.808,Z 1137.633,A -85,B 0,C 180,E1 2638.144,E2 2638.144} C_VEL
LIN {X 0,Y 115.676,Z 1148.934,A -85,B 0,C 180,E1 2635.397,E2 2635.397} C_VEL
LIN {X 0,Y 96.777,Z 1159.612,A -85,B 0,C 180,E1 2631.583,E2 2631.583} C_VEL
LIN {X 0,Y 73.08,Z 1171.565,A -85,B 0,C 180,E1 2624.258,E2 2624.258} C_VEL
LIN {X 0,Y 54.11,Z 1180.184,A -85,B 0,C 180,E1 2613.746,E2 2613.746} C_VEL
LIN {X 0,Y 39.886,Z 1186.697,A -85,B 0,C 180,E1 2597.871,E2 2597.871} C_VEL
LIN {X 0,Y 30.673,Z 1192.145,A -85,B 0,C 180,E1 2571.732,E2 2571.732} C_VEL
LIN {X 0,Y 28.835,Z 1196.242,A -85,B 0,C 180,E1 2542.423,E2 2542.423} C_VEL
LIN {X 0,Y 33.944,Z 1200.438,A -85,B 0,C 180,E1 2511.531,E2 2511.531} C_VEL
LIN {X 0,Y 41.976,Z 1203.37,A -85,B 0,C 180,E1 2494.843,E2 2494.843} C_VEL
LIN {X 0,Y 30.502,Z 1204.52,A -85,B 0,C 180,E1 2463.867,E2 2463.867} C_VEL
LIN {X 0,Y 30.345,Z 1204.697,A -85,B 0,C 180,E1 2429.999,E2 2429.999} C_VEL
LIN {X 0,Y 31.252,Z 1201.554,A -85,B 0,C 180,E1 2394.838,E2 2394.838} C_VEL
LIN {X 0,Y 44.708,Z 1195.666,A -85,B 0,C 180,E1 2363.516,E2 2363.516} C_VEL
LIN {X 0,Y 60.936,Z 1189.314,A -85,B 0,C 180,E1 2350.096,E2 2350.096} C_VEL
LIN {X 0,Y 78.068,Z 1182.042,A -85,B 0,C 180,E1 2342.557,E2 2342.557} C_VEL
LIN {X 0,Y 96.073,Z 1173.481,A -85,B 0,C 180,E1 2337.597,E2 2337.597} C_VEL
LIN {X 0,Y 115.628,Z 1163.015,A -85,B 0,C 180,E1 2333.959,E2 2333.959} C_VEL
LIN {X 0,Y 139.775,Z 1148.157,A -85,B 0,C 180,E1 2330.815,E2 2330.815} C_VEL
LIN {X 0,Y 158.039,Z 1135.388,A -85,B 0,C 180,E1 2329.058,E2 2329.058} C_VEL
LIN {X 0,Y 176.035,Z 1121.438,A -85,B 0,C 180,E1 2327.676,E2 2327.676} C_VEL
LIN {X 0,Y 197.023,Z 1103.32,A -85,B 0,C 180,E1 2326.372,E2 2326.372} C_VEL
LIN {X 0,Y 215.919,Z 1084.765,A -85,B 0,C 180,E1 2325.429,E2 2325.429} C_VEL
LIN {X 0,Y 231.064,Z 1068.382,A -85,B 0,C 180,E1 2324.793,E2 2324.793} C_VEL
LIN {X 0,Y 248.386,Z 1047.73,A -85,B 0,C 180,E1 2324.174,E2 2324.174} C_VEL
LIN {X 0,Y 265.707,Z 1024.302,A -85,B 0,C 180,E1 2323.655,E2 2323.655} C_VEL
LIN {X 0,Y 279.215,Z 1003.93,A -85,B 0,C 180,E1 2323.32,E2 2323.32} C_VEL
LIN {X 0,Y 294.343,Z 978.421,A -85,B 0,C 180,E1 2323.014,E2 2323.014} C_VEL
LIN {X 0,Y 307.179,Z 953.434,A -85,B 0,C 180,E1 2322.814,E2 2322.814} C_VEL
LIN {X 0,Y 318.704,Z 927.999,A -85,B 0,C 180,E1 2322.68,E2 2322.68} C_VEL
LIN {X 0,Y 329.097,Z 900.912,A -85,B 0,C 180,E1 2322.555,E2 2322.555} C_VEL
LIN {X 0,Y 337.043,Z 876.143,A -85,B 0,C 180,E1 2322.383,E2 2322.383} C_VEL
LIN {X 0,Y 341.846,Z 858.549,A -85,B 0,C 180,E1 2322.246,E2 2322.246} C_VEL
LIN {X 0,Y 343.574,Z 851.086,A -85,B 0,C 180,E1 2322.024,E2 2322.024} C_VEL
LIN {X 0,Y 346.853,Z 831.317,A -85,B 0,C 180,E1 2320.845,E2 2320.845} C_VEL
LIN {X 0,Y 348.029,Z 824.837,A -85,B 0,C 180,E1 2320.681,E2 2320.681} C_VEL
LIN {X 0,Y 356.304,Z 782.044,A -85,B 0,C 180,E1 2320.363,E2 2320.363} C_VEL
LIN {X 0,Y 354.944,Z 779.373,A -85,B 0,C 180,E1 2317.94,E2 2317.94} C_VEL
LIN {X 0,Y 352.404,Z 775.721,A -85,B 0,C 180,E1 2312.452,E2 2312.452} C_VEL
LIN {X 0,Y 352.032,Z 774.633,A -85,B 0,C 180,E1 2310.689,E2 2310.689} C_VEL
LIN {X 0,Y 351.164,Z 774.104,A -85,B 0,C 180,E1 2305.374,E2 2305.374} C_VEL
LIN {X 0,Y 351.859,Z 774.371,A -85,B 0,C 180,E1 2300.041,E2 2300.041} C_VEL
LIN {X 0,Y 352.876,Z 775.053,A -85,B 0,C 180,E1 2296.93,E2 2296.93} C_VEL
LIN {X 0,Y 354.452,Z 778.051,A -85,B 0,C 180,E1 2293.183,E2 2293.183} C_VEL
LIN {X 0,Y 344.209,Z 828.86,A -85,B 0,C 180,E1 2292.839,E2 2292.839} C_VEL
LIN {X 0,Y 336.54,Z 857.664,A -85,B 0,C 180,E1 2292.576,E2 2292.576} C_VEL
LIN {X 0,Y 327.674,Z 885.352,A -85,B 0,C 180,E1 2292.274,E2 2292.274} C_VEL
LIN {X 0,Y 316.737,Z 913.519,A -85,B 0,C 180,E1 2291.899,E2 2291.899} C_VEL
LIN {X 0,Y 306.179,Z 937.131,A -85,B 0,C 180,E1 2291.524,E2 2291.524} C_VEL
LIN {X 0,Y 291.452,Z 965.641,A -85,B 0,C 180,E1 2290.995,E2 2290.995} C_VEL
LIN {X 0,Y 278.599,Z 987.434,A -85,B 0,C 180,E1 2290.511,E2 2290.511} C_VEL
LIN {X 0,Y 262.762,Z 1011.501,A -85,B 0,C 180,E1 2289.88,E2 2289.88} C_VEL
LIN {X 0,Y 245.507,Z 1034.406,A -85,B 0,C 180,E1 2289.144,E2 2289.144} C_VEL
LIN {X 0,Y 230.066,Z 1052.92,A -85,B 0,C 180,E1 2288.425,E2 2288.425} C_VEL
LIN {X 0,Y 210.219,Z 1074.294,A -85,B 0,C 180,E1 2287.408,E2 2287.408} C_VEL
LIN {X 0,Y 191.557,Z 1092.083,A -85,B 0,C 180,E1 2286.322,E2 2286.322} C_VEL
LIN {X 0,Y 174.132,Z 1107.151,A -85,B 0,C 180,E1 2285.17,E2 2285.17} C_VEL
LIN {X 0,Y 152.185,Z 1124.241,A -85,B 0,C 180,E1 2283.444,E2 2283.444} C_VEL
LIN {X 0,Y 130.672,Z 1138.9,A -85,B 0,C 180,E1 2281.354,E2 2281.354} C_VEL
LIN {X 0,Y 112.077,Z 1150.278,A -85,B 0,C 180,E1 2279.037,E2 2279.037} C_VEL
LIN {X 0,Y 91.639,Z 1161.497,A -85,B 0,C 180,E1 2275.623,E2 2275.623} C_VEL
LIN {X 0,Y 66.63,Z 1173.557,A -85,B 0,C 180,E1 2269.015,E2 2269.015} C_VEL
LIN {X 0,Y 47.536,Z 1181.797,A -85,B 0,C 180,E1 2259.688,E2 2259.688} C_VEL
LIN {X 0,Y 32.205,Z 1188.177,A -85,B 0,C 180,E1 2243.478,E2 2243.478} C_VEL
LIN {X 0,Y 22.131,Z 1193.588,A -85,B 0,C 180,E1 2210.765,E2 2210.765} C_VEL
LIN {X 0,Y 21.533,Z 1197.693,A -85,B 0,C 180,E1 2170.705,E2 2170.705} C_VEL
LIN {X 0,Y 31.001,Z 1202.184,A -85,B 0,C 180,E1 2134.855,E2 2134.855} C_VEL
LIN {X 0,Y 21.556,Z 1202.796,A -85,B 0,C 180,E1 2083.074,E2 2083.074} C_VEL
LIN {X 0,Y 22.365,Z 1202.677,A -85,B 0,C 180,E1 2069.999,E2 2069.999} C_VEL
LIN {X 0,Y 25.602,Z 1199.088,A -85,B 0,C 180,E1 2021.601,E2 2021.601} C_VEL
LIN {X 0,Y 40.314,Z 1193.827,A -85,B 0,C 180,E1 1994.693,E2 1994.693} C_VEL
LIN {X 0,Y 57.096,Z 1187.766,A -85,B 0,C 180,E1 1983.434,E2 1983.434} C_VEL
LIN {X 0,Y 75.087,Z 1180.471,A -85,B 0,C 180,E1 1977.107,E2 1977.107} C_VEL
LIN {X 0,Y 92.901,Z 1172.277,A -85,B 0,C 180,E1 1973.2,E2 1973.2} C_VEL
LIN {X 0,Y 111.548,Z 1162.59,A -85,B 0,C 180,E1 1970.402,E2 1970.402} C_VEL
LIN {X 0,Y 134.259,Z 1149.182,A -85,B 0,C 180,E1 1967.964,E2 1967.964} C_VEL
LIN {X 0,Y 155.401,Z 1134.718,A -85,B 0,C 180,E1 1966.303,E2 1966.303} C_VEL
LIN {X 0,Y 172.682,Z 1121.559,A -85,B 0,C 180,E1 1965.235,E2 1965.235} C_VEL
LIN {X 0,Y 191.107,Z 1106.014,A -85,B 0,C 180,E1 1964.3,E2 1964.3} C_VEL
LIN {X 0,Y 212.835,Z 1085.295,A -85,B 0,C 180,E1 1963.409,E2 1963.409} C_VEL
LIN {X 0,Y 229.146,Z 1067.838,A -85,B 0,C 180,E1 1962.863,E2 1962.863} C_VEL
LIN {X 0,Y 245.453,Z 1048.57,A -85,B 0,C 180,E1 1962.405,E2 1962.405} C_VEL
LIN {X 0,Y 263.931,Z 1023.908,A -85,B 0,C 180,E1 1961.969,E2 1961.969} C_VEL
LIN {X 0,Y 277.288,Z 1003.904,A -85,B 0,C 180,E1 1961.716,E2 1961.716} C_VEL
LIN {X 0,Y 292.069,Z 979.269,A -85,B 0,C 180,E1 1961.494,E2 1961.494} C_VEL
LIN {X 0,Y 305.314,Z 953.732,A -85,B 0,C 180,E1 1961.35,E2 1961.35} C_VEL
LIN {X 0,Y 316.205,Z 929.937,A -85,B 0,C 180,E1 1961.272,E2 1961.272} C_VEL
LIN {X 0,Y 327.457,Z 901.182,A -85,B 0,C 180,E1 1961.186,E2 1961.186} C_VEL
LIN {X 0,Y 335.597,Z 876.035,A -85,B 0,C 180,E1 1961.043,E2 1961.043} C_VEL
LIN {X 0,Y 343.246,Z 847.463,A -85,B 0,C 180,E1 1960.839,E2 1960.839} C_VEL
LIN {X 0,Y 348.029,Z 824.837,A -85,B 0,C 180,E1 1960.681,E2 1960.681} C_VEL
LIN {X 0,Y 349.345,Z 817.292,A -85,B 0,C 180,E1 1960.471,E2 1960.471} C_VEL
LIN {X 0,Y 352.335,Z 797.437,A -85,B 0,C 180,E1 1959.334,E2 1959.334} C_VEL
LIN {X 0,Y 353.504,Z 790.956,A -85,B 0,C 180,E1 1959.172,E2 1959.172} C_VEL
LIN {X 0,Y 353.995,Z 788.431,A -85,B 0,C 180,E1 1959.151,E2 1959.151} C_VEL
LIN {X 0,Y 353.005,Z 786.949,A -85,B 0,C 180,E1 1957.426,E2 1957.426} C_VEL
LIN {X 0,Y 350.703,Z 783.222,A -85,B 0,C 180,E1 1951.937,E2 1951.937} C_VEL
LIN {X 0,Y 350.357,Z 782.43,A -85,B 0,C 180,E1 1950.414,E2 1950.414} C_VEL
LIN {X 0,Y 349.592,Z 781.938,A -85,B 0,C 180,E1 1945.108,E2 1945.108} C_VEL
LIN {X 0,Y 350.38,Z 782.265,A -85,B 0,C 180,E1 1939.624,E2 1939.624} C_VEL
LIN {X 0,Y 351.305,Z 782.973,A -85,B 0,C 180,E1 1936.914,E2 1936.914} C_VEL
LIN {X 0,Y 352.202,Z 785.024,A -85,B 0,C 180,E1 1934.432,E2 1934.432} C_VEL
LIN {X 0,Y 342.776,Z 830.928,A -85,B 0,C 180,E1 1934.147,E2 1934.147} C_VEL
LIN {X 0,Y 335.21,Z 859.091,A -85,B 0,C 180,E1 1933.919,E2 1933.919} C_VEL
LIN {X 0,Y 325.969,Z 887.677,A -85,B 0,C 180,E1 1933.643,E2 1933.643} C_VEL
LIN {X 0,Y 315.185,Z 915.097,A -85,B 0,C 180,E1 1933.319,E2 1933.319} C_VEL
LIN {X 0,Y 303.997,Z 939.884,A -85,B 0,C 180,E1 1932.974,E2 1932.974} C_VEL
LIN {X 0,Y 289.87,Z 966.917,A -85,B 0,C 180,E1 1932.538,E2 1932.538} C_VEL
LIN {X 0,Y 276.796,Z 988.95,A -85,B 0,C 180,E1 1932.118,E2 1932.118} C_VEL
LIN {X 0,Y 260.64,Z 1013.281,A -85,B 0,C 180,E1 1931.575,E2 1931.575} C_VEL
LIN {X 0,Y 243.654,Z 1035.686,A -85,B 0,C 180,E1 1930.967,E2 1930.967} C_VEL
LIN {X 0,Y 227.771,Z 1054.612,A -85,B 0,C 180,E1 1930.354,E2 1930.354} C_VEL
LIN {X 0,Y 206.191,Z 1077.472,A -85,B 0,C 180,E1 1929.439,E2 1929.439} C_VEL
LIN {X 0,Y 189.02,Z 1093.675,A -85,B 0,C 180,E1 1928.623,E2 1928.623} C_VEL
LIN {X 0,Y 170.462,Z 1109.527,A -85,B 0,C 180,E1 1927.638,E2 1927.638} C_VEL
LIN {X 0,Y 146.553,Z 1127.595,A -85,B 0,C 180,E1 1926.14,E2 1926.14} C_VEL
LIN {X 0,Y 127.688,Z 1140.212,A -85,B 0,C 180,E1 1924.691,E2 1924.691} C_VEL
LIN {X 0,Y 108.679,Z 1151.668,A -85,B 0,C 180,E1 1922.876,E2 1922.876} C_VEL
LIN {X 0,Y 86.648,Z 1163.549,A -85,B 0,C 180,E1 1920.062,E2 1920.062} C_VEL
LIN {X 0,Y 61.542,Z 1175.197,A -85,B 0,C 180,E1 1914.988,E2 1914.988} C_VEL
LIN {X 0,Y 41.966,Z 1183.175,A -85,B 0,C 180,E1 1907.625,E2 1907.625} C_VEL
LIN {X 0,Y 24.891,Z 1189.691,A -85,B 0,C 180,E1 1892.303,E2 1892.303} C_VEL
LIN {X 0,Y 13.848,Z 1194.733,A -85,B 0,C 180,E1 1852.588,E2 1852.588} C_VEL
LIN {X 0,Y 15.261,Z 1198.818,A -85,B 0,C 180,E1 1792.471,E2 1792.471} C_VEL
LIN {X 0,Y 19.676,Z 1200.573,A -85,B 0,C 180,E1 1773.843,E2 1773.843} C_VEL
LIN {X 0,Y 14.337,Z 1200.602,A -85,B 0,C 180,E1 1709.998,E2 1709.998} C_VEL
LIN {X 0,Y 19.464,Z 1197.291,A -85,B 0,C 180,E1 1649.151,E2 1649.151} C_VEL
LIN {X 0,Y 36.119,Z 1192.246,A -85,B 0,C 180,E1 1624.73,E2 1624.73} C_VEL
LIN {X 0,Y 54.554,Z 1186.05,A -85,B 0,C 180,E1 1615.795,E2 1615.795} C_VEL
LIN {X 0,Y 73.889,Z 1178.482,A -85,B 0,C 180,E1 1611.06,E2 1611.06} C_VEL
LIN {X 0,Y 94.019,Z 1169.321,A -85,B 0,C 180,E1 1608.071,E2 1608.071} C_VEL
LIN {X 0,Y 118.687,Z 1156.155,A -85,B 0,C 180,E1 1605.654,E2 1605.654} C_VEL
LIN {X 0,Y 138.137,Z 1144.159,A -85,B 0,C 180,E1 1604.301,E2 1604.301} C_VEL
LIN {X 0,Y 156.588,Z 1131.42,A -85,B 0,C 180,E1 1603.297,E2 1603.297} C_VEL
LIN {X 0,Y 177.277,Z 1115.467,A -85,B 0,C 180,E1 1602.4,E2 1602.4} C_VEL
LIN {X 0,Y 198.546,Z 1096.702,A -85,B 0,C 180,E1 1601.674,E2 1601.674} C_VEL
LIN {X 0,Y 215.474,Z 1080.05,A -85,B 0,C 180,E1 1601.197,E2 1601.197} C_VEL
LIN {X 0,Y 234.588,Z 1059.191,A -85,B 0,C 180,E1 1600.75,E2 1600.75} C_VEL
LIN {X 0,Y 252.044,Z 1037.464,A -85,B 0,C 180,E1 1600.421,E2 1600.421} C_VEL
LIN {X 0,Y 266.735,Z 1017.194,A -85,B 0,C 180,E1 1600.202,E2 1600.202} C_VEL
LIN {X 0,Y 284.097,Z 990.102,A -85,B 0,C 180,E1 1600.002,E2 1600.002} C_VEL
LIN {X 0,Y 296.513,Z 967.99,A -85,B 0,C 180,E1 1599.907,E2 1599.907} C_VEL
LIN {X 0,Y 309.5,Z 941.93,A -85,B 0,C 180,E1 1599.846,E2 1599.846} C_VEL
LIN {X 0,Y 320.891,Z 914.972,A -85,B 0,C 180,E1 1599.833,E2 1599.833} C_VEL
LIN {X 0,Y 329.275,Z 891.943,A -85,B 0,C 180,E1 1599.769,E2 1599.769} C_VEL
LIN {X 0,Y 338.509,Z 861.235,A -85,B 0,C 180,E1 1599.607,E2 1599.607} C_VEL
LIN {X 0,Y 344.659,Z 835.447,A -85,B 0,C 180,E1 1599.442,E2 1599.442} C_VEL
LIN {X 0,Y 353.504,Z 790.956,A -85,B 0,C 180,E1 1599.172,E2 1599.172} C_VEL
LIN {X 0,Y 353.67,Z 789.464,A -85,B 0,C 180,E1 1598.989,E2 1598.989} C_VEL
LIN {X 0,Y 353.454,Z 788.78,A -85,B 0,C 180,E1 1598.496,E2 1598.496} C_VEL
LIN {X 0,Y 352.702,Z 789.609,A -85,B 0,C 180,E1 1597.719,E2 1597.719} C_VEL
LIN {X 0,Y 350.829,Z 793.166,A -85,B 0,C 180,E1 1596.094,E2 1596.094} C_VEL
LIN {X 0,Y 350.312,Z 793.489,A -85,B 0,C 180,E1 1595.32,E2 1595.32} C_VEL
LIN {X 0,Y 348.848,Z 790.307,A -85,B 0,C 180,E1 1590.614,E2 1590.614} C_VEL
LIN {X 0,Y 348.014,Z 789.787,A -85,B 0,C 180,E1 1585.256,E2 1585.256} C_VEL
LIN {X 0,Y 348.77,Z 790.086,A -85,B 0,C 180,E1 1579.83,E2 1579.83} C_VEL
LIN {X 0,Y 349.681,Z 790.76,A -85,B 0,C 180,E1 1577.055,E2 1577.055} C_VEL
LIN {X 0,Y 350.111,Z 791.908,A -85,B 0,C 180,E1 1575.698,E2 1575.698} C_VEL
LIN {X 0,Y 341.501,Z 833.084,A -85,B 0,C 180,E1 1575.465,E2 1575.465} C_VEL
LIN {X 0,Y 334.098,Z 860.391,A -85,B 0,C 180,E1 1575.273,E2 1575.273} C_VEL
LIN {X 0,Y 324.72,Z 889.171,A -85,B 0,C 180,E1 1575.032,E2 1575.032} C_VEL
LIN {X 0,Y 313.856,Z 916.607,A -85,B 0,C 180,E1 1574.753,E2 1574.753} C_VEL
LIN {X 0,Y 302.603,Z 941.387,A -85,B 0,C 180,E1 1574.461,E2 1574.461} C_VEL
LIN {X 0,Y 288.772,Z 967.722,A -85,B 0,C 180,E1 1574.104,E2 1574.104} C_VEL
LIN {X 0,Y 276.073,Z 989.096,A -85,B 0,C 180,E1 1573.77,E2 1573.77} C_VEL
LIN {X 0,Y 260.305,Z 1012.908,A -85,B 0,C 180,E1 1573.34,E2 1573.34} C_VEL
LIN {X 0,Y 242.658,Z 1036.172,A -85,B 0,C 180,E1 1572.835,E2 1572.835} C_VEL
LIN {X 0,Y 227.042,Z 1054.722,A -85,B 0,C 180,E1 1572.361,E2 1572.361} C_VEL
LIN {X 0,Y 207.329,Z 1075.785,A -85,B 0,C 180,E1 1571.723,E2 1571.723} C_VEL
LIN {X 0,Y 188.254,Z 1093.789,A -85,B 0,C 180,E1 1571.043,E2 1571.043} C_VEL
LIN {X 0,Y 170.586,Z 1108.887,A -85,B 0,C 180,E1 1570.359,E2 1570.359} C_VEL
LIN {X 0,Y 148.805,Z 1125.69,A -85,B 0,C 180,E1 1569.399,E2 1569.399} C_VEL
LIN {X 0,Y 126.008,Z 1140.977,A -85,B 0,C 180,E1 1568.225,E2 1568.225} C_VEL
LIN {X 0,Y 106.367,Z 1152.745,A -85,B 0,C 180,E1 1566.986,E2 1566.986} C_VEL
LIN {X 0,Y 83.108,Z 1165.072,A -85,B 0,C 180,E1 1565.102,E2 1565.102} C_VEL
LIN {X 0,Y 57.807,Z 1176.526,A -85,B 0,C 180,E1 1562.053,E2 1562.053} C_VEL
LIN {X 0,Y 37.259,Z 1184.634,A -85,B 0,C 180,E1 1557.675,E2 1557.675} C_VEL
LIN {X 0,Y 18.934,Z 1191.023,A -85,B 0,C 180,E1 1548.086,E2 1548.086} C_VEL
LIN {X 0,Y 5.664,Z 1195.798,A -85,B 0,C 180,E1 1501.972,E2 1501.972} C_VEL
LIN {X 0,Y 8.219,Z 1198.609,A -85,B 0,C 180,E1 1410.084,E2 1410.084} C_VEL
LIN {X 0,Y 6.312,Z 1198.491,A -85,B 0,C 180,E1 1349.997,E2 1349.997} C_VEL
LIN {X 0,Y 16.078,Z 1195.235,A -85,B 0,C 180,E1 1265.702,E2 1265.702} C_VEL
LIN {X 0,Y 33.271,Z 1190.653,A -85,B 0,C 180,E1 1252.633,E2 1252.633} C_VEL
LIN {X 0,Y 52.185,Z 1184.578,A -85,B 0,C 180,E1 1247.736,E2 1247.736} C_VEL
LIN {X 0,Y 71.383,Z 1177.261,A -85,B 0,C 180,E1 1245.126,E2 1245.126} C_VEL
LIN {X 0,Y 91.106,Z 1168.506,A -85,B 0,C 180,E1 1243.42,E2 1243.42} C_VEL
LIN {X 0,Y 116.104,Z 1155.489,A -85,B 0,C 180,E1 1241.939,E2 1241.939} C_VEL
LIN {X 0,Y 136.36,Z 1143.18,A -85,B 0,C 180,E1 1241.069,E2 1241.069} C_VEL
LIN {X 0,Y 153.832,Z 1131.276,A -85,B 0,C 180,E1 1240.47,E2 1240.47} C_VEL
LIN {X 0,Y 172.43,Z 1117.16,A -85,B 0,C 180,E1 1239.951,E2 1239.951} C_VEL
LIN {X 0,Y 195.427,Z 1097.393,A -85,B 0,C 180,E1 1239.438,E2 1239.438} C_VEL
LIN {X 0,Y 212.955,Z 1080.356,A -85,B 0,C 180,E1 1239.124,E2 1239.124} C_VEL
LIN {X 0,Y 229.382,Z 1062.702,A -85,B 0,C 180,E1 1238.88,E2 1238.88} C_VEL
LIN {X 0,Y 249.068,Z 1038.898,A -85,B 0,C 180,E1 1238.647,E2 1238.647} C_VEL
LIN {X 0,Y 263.893,Z 1018.697,A -85,B 0,C 180,E1 1238.521,E2 1238.521} C_VEL
LIN {X 0,Y 279.556,Z 994.956,A -85,B 0,C 180,E1 1238.424,E2 1238.424} C_VEL
LIN {X 0,Y 294.158,Z 969.49,A -85,B 0,C 180,E1 1238.382,E2 1238.382} C_VEL
LIN {X 0,Y 305.99,Z 946.187,A -85,B 0,C 180,E1 1238.381,E2 1238.381} C_VEL
LIN {X 0,Y 318.819,Z 916.916,A -85,B 0,C 180,E1 1238.416,E2 1238.416} C_VEL
LIN {X 0,Y 327.315,Z 894.073,A -85,B 0,C 180,E1 1238.396,E2 1238.396} C_VEL
LIN {X 0,Y 335.807,Z 867.173,A -85,B 0,C 180,E1 1238.292,E2 1238.292} C_VEL
LIN {X 0,Y 343.101,Z 837.869,A -85,B 0,C 180,E1 1238.134,E2 1238.134} C_VEL
LIN {X 0,Y 351.733,Z 795.051,A -85,B 0,C 180,E1 1237.873,E2 1237.873} C_VEL
LIN {X 0,Y 350.312,Z 793.489,A -85,B 0,C 180,E1 1235.32,E2 1235.32} C_VEL
LIN {X 0,Y 349.655,Z 793.561,A -85,B 0,C 180,E1 1234.053,E2 1234.053} C_VEL
LIN {X 0,Y 347.218,Z 797.813,A -85,B 0,C 180,E1 1230.265,E2 1230.265} C_VEL
LIN {X 0,Y 346.944,Z 797.978,A -85,B 0,C 180,E1 1229.528,E2 1229.528} C_VEL
LIN {X 0,Y 346.512,Z 797.602,A -85,B 0,C 180,E1 1224.142,E2 1224.142} C_VEL
LIN {X 0,Y 347.618,Z 798.117,A -85,B 0,C 180,E1 1218.36,E2 1218.36} C_VEL
LIN {X 0,Y 348.132,Z 798.731,A -85,B 0,C 180,E1 1216.975,E2 1216.975} C_VEL
LIN {X 0,Y 339.718,Z 837.532,A -85,B 0,C 180,E1 1216.78,E2 1216.78} C_VEL
LIN {X 0,Y 332.568,Z 863.372,A -85,B 0,C 180,E1 1216.622,E2 1216.622} C_VEL
LIN {X 0,Y 322.688,Z 892.885,A -85,B 0,C 180,E1 1216.411,E2 1216.411} C_VEL
LIN {X 0,Y 312.485,Z 918.368,A -85,B 0,C 180,E1 1216.196,E2 1216.196} C_VEL
LIN {X 0,Y 300.204,Z 945.127,A -85,B 0,C 180,E1 1215.938,E2 1215.938} C_VEL
LIN {X 0,Y 286.623,Z 970.442,A -85,B 0,C 180,E1 1215.654,E2 1215.654} C_VEL
LIN {X 0,Y 273.317,Z 992.543,A -85,B 0,C 180,E1 1215.379,E2 1215.379} C_VEL
LIN {X 0,Y 255.424,Z 1018.779,A -85,B 0,C 180,E1 1215.004,E2 1215.004} C_VEL
LIN {X 0,Y 240.318,Z 1038.41,A -85,B 0,C 180,E1 1214.68,E2 1214.68} C_VEL
LIN {X 0,Y 223.315,Z 1058.407,A -85,B 0,C 180,E1 1214.305,E2 1214.305} C_VEL
LIN {X 0,Y 202.852,Z 1079.737,A -85,B 0,C 180,E1 1213.835,E2 1213.835} C_VEL
LIN {X 0,Y 185.482,Z 1095.959,A -85,B 0,C 180,E1 1213.418,E2 1213.418} C_VEL
LIN {X 0,Y 166.677,Z 1111.87,A -85,B 0,C 180,E1 1212.956,E2 1212.956} C_VEL
LIN {X 0,Y 142.535,Z 1129.915,A -85,B 0,C 180,E1 1212.333,E2 1212.333} C_VEL
LIN {X 0,Y 123.033,Z 1142.761,A -85,B 0,C 180,E1 1211.79,E2 1211.79} C_VEL
LIN {X 0,Y 103.178,Z 1154.499,A -85,B 0,C 180,E1 1211.222,E2 1211.222} C_VEL
LIN {X 0,Y 78.91,Z 1167.243,A -85,B 0,C 180,E1 1210.511,E2 1210.511} C_VEL
LIN {X 0,Y 54.492,Z 1178.069,A -85,B 0,C 180,E1 1209.958,E2 1209.958} C_VEL
LIN {X 0,Y 34.008,Z 1185.99,A -85,B 0,C 180,E1 1210.141,E2 1210.141} C_VEL
LIN {X 0,Y 15.343,Z 1192.407,A -85,B 0,C 180,E1 1214.204,E2 1214.204} C_VEL
LIN {X 0,Y 6.812,Z 1195.238,A -85,B 0,C 180,E1 1229.588,E2 1229.588} C_VEL
LIN {X 0,Y 27.88,Z 1190.205,A -85,B 0,C 180,E1 1238.82,E2 1238.82} C_VEL
LIN {X 0,Y 48.156,Z 1184.045,A -85,B 0,C 180,E1 1239.125,E2 1239.125} C_VEL
LIN {X 0,Y 67.531,Z 1176.933,A -85,B 0,C 180,E1 1238.874,E2 1238.874} C_VEL
LIN {X 0,Y 85.946,Z 1168.998,A -85,B 0,C 180,E1 1238.545,E2 1238.545} C_VEL
LIN {X 0,Y 104.429,Z 1159.881,A -85,B 0,C 180,E1 1238.24,E2 1238.24} C_VEL
LIN {X 0,Y 125.167,Z 1148.237,A -85,B 0,C 180,E1 1237.918,E2 1237.918} C_VEL
LIN {X 0,Y 149.443,Z 1132.411,A -85,B 0,C 180,E1 1237.581,E2 1237.581} C_VEL
LIN {X 0,Y 167.906,Z 1118.719,A -85,B 0,C 180,E1 1237.372,E2 1237.372} C_VEL
LIN {X 0,Y 185.776,Z 1103.992,A -85,B 0,C 180,E1 1237.2,E2 1237.2} C_VEL
LIN {X 0,Y 207.429,Z 1083.953,A -85,B 0,C 180,E1 1237.026,E2 1237.026} C_VEL
LIN {X 0,Y 224.975,Z 1065.557,A -85,B 0,C 180,E1 1236.924,E2 1236.924} C_VEL
LIN {X 0,Y 240.808,Z 1047.173,A -85,B 0,C 180,E1 1236.861,E2 1236.861} C_VEL
LIN {X 0,Y 259.44,Z 1022.835,A -85,B 0,C 180,E1 1236.805,E2 1236.805} C_VEL
LIN {X 0,Y 274.138,Z 1001.084,A -85,B 0,C 180,E1 1236.8,E2 1236.8} C_VEL
LIN {X 0,Y 288.687,Z 977.036,A -85,B 0,C 180,E1 1236.824,E2 1236.824} C_VEL
LIN {X 0,Y 302.237,Z 951.18,A -85,B 0,C 180,E1 1236.882,E2 1236.882} C_VEL
LIN {X 0,Y 312.939,Z 927.99,A -85,B 0,C 180,E1 1236.954,E2 1236.954} C_VEL
LIN {X 0,Y 324.262,Z 899.454,A -85,B 0,C 180,E1 1237.011,E2 1237.011} C_VEL
LIN {X 0,Y 332.648,Z 873.899,A -85,B 0,C 180,E1 1236.962,E2 1236.962} C_VEL
LIN {X 0,Y 340.225,Z 846.144,A -85,B 0,C 180,E1 1236.846,E2 1236.846} C_VEL
LIN {X 0,Y 349.363,Z 802.217,A -85,B 0,C 180,E1 1236.636,E2 1236.636} C_VEL
LIN {X 0,Y 347.299,Z 798.166,A -85,B 0,C 180,E1 1230.696,E2 1230.696} C_VEL
LIN {X 0,Y 346.944,Z 797.978,A -85,B 0,C 180,E1 1229.528,E2 1229.528} C_VEL
LIN {X 0,Y 346.525,Z 798.778,A -85,B 0,C 180,E1 1228.254,E2 1228.254} C_VEL
LIN {X 0,Y 345.011,Z 804.895,A -85,B 0,C 180,E1 1224.694,E2 1224.694} C_VEL
LIN {X 0,Y 344.984,Z 805.458,A -85,B 0,C 180,E1 1223.774,E2 1223.774} C_VEL
LIN {X 0,Y 346.082,Z 805.981,A -85,B 0,C 180,E1 1218.269,E2 1218.269} C_VEL
LIN {X 0,Y 338.601,Z 839.605,A -85,B 0,C 180,E1 1218.119,E2 1218.119} C_VEL
LIN {X 0,Y 331.348,Z 865.556,A -85,B 0,C 180,E1 1217.987,E2 1217.987} C_VEL
LIN {X 0,Y 320.847,Z 896.332,A -85,B 0,C 180,E1 1217.807,E2 1217.807} C_VEL
LIN {X 0,Y 311.181,Z 920.24,A -85,B 0,C 180,E1 1217.649,E2 1217.649} C_VEL
LIN {X 0,Y 298.606,Z 947.358,A -85,B 0,C 180,E1 1217.448,E2 1217.448} C_VEL
LIN {X 0,Y 285.312,Z 971.99,A -85,B 0,C 180,E1 1217.239,E2 1217.239} C_VEL
LIN {X 0,Y 271.887,Z 994.197,A -85,B 0,C 180,E1 1217.04,E2 1217.04} C_VEL
LIN {X 0,Y 253.84,Z 1020.491,A -85,B 0,C 180,E1 1216.779,E2 1216.779} C_VEL
LIN {X 0,Y 238.23,Z 1040.668,A -85,B 0,C 180,E1 1216.56,E2 1216.56} C_VEL
LIN {X 0,Y 219.853,Z 1062.095,A -85,B 0,C 180,E1 1216.313,E2 1216.313} C_VEL
LIN {X 0,Y 199.954,Z 1082.423,A -85,B 0,C 180,E1 1216.061,E2 1216.061} C_VEL
LIN {X 0,Y 181.912,Z 1099.036,A -85,B 0,C 180,E1 1215.854,E2 1215.854} C_VEL
LIN {X 0,Y 159.399,Z 1117.607,A -85,B 0,C 180,E1 1215.651,E2 1215.651} C_VEL
LIN {X 0,Y 138.46,Z 1132.779,A -85,B 0,C 180,E1 1215.533,E2 1215.533} C_VEL
LIN {X 0,Y 119.882,Z 1144.918,A -85,B 0,C 180,E1 1215.523,E2 1215.523} C_VEL
LIN {X 0,Y 98.839,Z 1157.261,A -85,B 0,C 180,E1 1215.731,E2 1215.731} C_VEL
LIN {X 0,Y 72.363,Z 1170.684,A -85,B 0,C 180,E1 1216.683,E2 1216.683} C_VEL
LIN {X 0,Y 51.31,Z 1179.968,A -85,B 0,C 180,E1 1218.887,E2 1218.887} C_VEL
LIN {X 0,Y 32.024,Z 1187.585,A -85,B 0,C 180,E1 1224.797,E2 1224.797} C_VEL
LIN {X 0,Y 50.684,Z 1181.606,A -85,B 0,C 180,E1 1230.229,E2 1230.229} C_VEL
LIN {X 0,Y 71.031,Z 1173.887,A -85,B 0,C 180,E1 1232.478,E2 1232.478} C_VEL
LIN {X 0,Y 95.927,Z 1162.64,A -85,B 0,C 180,E1 1233.689,E2 1233.689} C_VEL
LIN {X 0,Y 117.728,Z 1150.914,A -85,B 0,C 180,E1 1234.194,E2 1234.194} C_VEL
LIN {X 0,Y 136.321,Z 1139.545,A -85,B 0,C 180,E1 1234.445,E2 1234.445} C_VEL
LIN {X 0,Y 156.273,Z 1125.833,A -85,B 0,C 180,E1 1234.615,E2 1234.615} C_VEL
LIN {X 0,Y 179.53,Z 1107.546,A -85,B 0,C 180,E1 1234.746,E2 1234.746} C_VEL
LIN {X 0,Y 197.421,Z 1091.658,A -85,B 0,C 180,E1 1234.821,E2 1234.821} C_VEL
LIN {X 0,Y 215.336,Z 1074.018,A -85,B 0,C 180,E1 1234.884,E2 1234.884} C_VEL
LIN {X 0,Y 235.62,Z 1051.411,A -85,B 0,C 180,E1 1234.959,E2 1234.959} C_VEL
LIN {X 0,Y 250.953,Z 1032.222,A -85,B 0,C 180,E1 1235.017,E2 1235.017} C_VEL
LIN {X 0,Y 267.859,Z 1008.711,A -85,B 0,C 180,E1 1235.105,E2 1235.105} C_VEL
LIN {X 0,Y 283.053,Z 984.447,A -85,B 0,C 180,E1 1235.209,E2 1235.209} C_VEL
LIN {X 0,Y 296,Z 961.266,A -85,B 0,C 180,E1 1235.322,E2 1235.322} C_VEL
LIN {X 0,Y 309.404,Z 933.584,A -85,B 0,C 180,E1 1235.464,E2 1235.464} C_VEL
LIN {X 0,Y 319.54,Z 909.266,A -85,B 0,C 180,E1 1235.584,E2 1235.584} C_VEL
LIN {X 0,Y 329.375,Z 881.594,A -85,B 0,C 180,E1 1235.603,E2 1235.603} C_VEL
LIN {X 0,Y 337.236,Z 854.236,A -85,B 0,C 180,E1 1235.537,E2 1235.537} C_VEL
LIN {X 0,Y 343.768,Z 826.269,A -85,B 0,C 180,E1 1235.427,E2 1235.427} C_VEL
LIN {X 0,Y 347.16,Z 809.264,A -85,B 0,C 180,E1 1235.343,E2 1235.343} C_VEL
LIN {X 0,Y 345.665,Z 805.982,A -85,B 0,C 180,E1 1230.537,E2 1230.537} C_VEL
LIN {X 0,Y 344.866,Z 805.469,A -85,B 0,C 180,E1 1225.135,E2 1225.135} C_VEL
LIN {X 0,Y 344.984,Z 805.458,A -85,B 0,C 180,E1 1223.774,E2 1223.774} C_VEL
LIN {X 0,Y 344.911,Z 806.507,A -85,B 0,C 180,E1 1222.923,E2 1222.923} C_VEL
LIN {X 0,Y 344.05,Z 812.777,A -85,B 0,C 180,E1 1220.758,E2 1220.758} C_VEL
LIN {X 0,Y 344.034,Z 813.602,A -85,B 0,C 180,E1 1220.022,E2 1220.022} C_VEL
LIN {X 0,Y 344.104,Z 813.787,A -85,B 0,C 180,E1 1219.562,E2 1219.562} C_VEL
LIN {X 0,Y 337.326,Z 842.997,A -85,B 0,C 180,E1 1219.46,E2 1219.46} C_VEL
LIN {X 0,Y 329.222,Z 871.384,A -85,B 0,C 180,E1 1219.345,E2 1219.345} C_VEL
LIN {X 0,Y 319.207,Z 899.757,A -85,B 0,C 180,E1 1219.219,E2 1219.219} C_VEL
LIN {X 0,Y 308.988,Z 924.65,A -85,B 0,C 180,E1 1219.102,E2 1219.102} C_VEL
LIN {X 0,Y 295.41,Z 953,A -85,B 0,C 180,E1 1218.955,E2 1218.955} C_VEL
LIN {X 0,Y 282.932,Z 975.729,A -85,B 0,C 180,E1 1218.828,E2 1218.828} C_VEL
LIN {X 0,Y 267.076,Z 1001.343,A -85,B 0,C 180,E1 1218.689,E2 1218.689} C_VEL
LIN {X 0,Y 250.815,Z 1024.325,A -85,B 0,C 180,E1 1218.565,E2 1218.565} C_VEL
LIN {X 0,Y 235.083,Z 1044.362,A -85,B 0,C 180,E1 1218.467,E2 1218.467} C_VEL
LIN {X 0,Y 214.663,Z 1067.469,A -85,B 0,C 180,E1 1218.382,E2 1218.382} C_VEL
LIN {X 0,Y 198.029,Z 1084.284,A -85,B 0,C 180,E1 1218.355,E2 1218.355} C_VEL
LIN {X 0,Y 180.564,Z 1100.345,A -85,B 0,C 180,E1 1218.38,E2 1218.38} C_VEL
LIN {X 0,Y 157.419,Z 1119.379,A -85,B 0,C 180,E1 1218.547,E2 1218.547} C_VEL
LIN {X 0,Y 136.715,Z 1134.383,A -85,B 0,C 180,E1 1218.877,E2 1218.877} C_VEL
LIN {X 0,Y 116.926,Z 1147.214,A -85,B 0,C 180,E1 1219.465,E2 1219.465} C_VEL
LIN {X 0,Y 92.896,Z 1161.131,A -85,B 0,C 180,E1 1220.802,E2 1220.802} C_VEL
LIN {X 0,Y 69.644,Z 1172.792,A -85,B 0,C 180,E1 1223.513,E2 1223.513} C_VEL
LIN {X 0,Y 63.689,Z 1175.595,A -85,B 0,C 180,E1 1224.723,E2 1224.723} C_VEL
LIN {X 0,Y 83.869,Z 1166.95,A -85,B 0,C 180,E1 1227.829,E2 1227.829} C_VEL
LIN {X 0,Y 102.336,Z 1157.889,A -85,B 0,C 180,E1 1229.464,E2 1229.464} C_VEL
LIN {X 0,Y 122.134,Z 1146.87,A -85,B 0,C 180,E1 1230.58,E2 1230.58} C_VEL
LIN {X 0,Y 146.82,Z 1131.032,A -85,B 0,C 180,E1 1231.464,E2 1231.464} C_VEL
LIN {X 0,Y 165.833,Z 1117.057,A -85,B 0,C 180,E1 1231.946,E2 1231.946} C_VEL
LIN {X 0,Y 183.522,Z 1102.602,A -85,B 0,C 180,E1 1232.294,E2 1232.294} C_VEL
LIN {X 0,Y 203.822,Z 1084.121,A -85,B 0,C 180,E1 1232.613,E2 1232.613} C_VEL
LIN {X 0,Y 222.845,Z 1064.306,A -85,B 0,C 180,E1 1232.875,E2 1232.875} C_VEL
LIN {X 0,Y 238.858,Z 1045.806,A -85,B 0,C 180,E1 1233.079,E2 1233.079} C_VEL
LIN {X 0,Y 257.151,Z 1022.145,A -85,B 0,C 180,E1 1233.288,E2 1233.288} C_VEL
LIN {X 0,Y 272.265,Z 999.92,A -85,B 0,C 180,E1 1233.475,E2 1233.475} C_VEL
LIN {X 0,Y 286.168,Z 977.107,A -85,B 0,C 180,E1 1233.657,E2 1233.657} C_VEL
LIN {X 0,Y 300.171,Z 950.798,A -85,B 0,C 180,E1 1233.859,E2 1233.859} C_VEL
LIN {X 0,Y 310.847,Z 927.88,A -85,B 0,C 180,E1 1234.033,E2 1234.033} C_VEL
LIN {X 0,Y 321.783,Z 901,A -85,B 0,C 180,E1 1234.188,E2 1234.188} C_VEL
LIN {X 0,Y 330.978,Z 873.404,A -85,B 0,C 180,E1 1234.216,E2 1234.216} C_VEL
LIN {X 0,Y 338.082,Z 847.854,A -85,B 0,C 180,E1 1234.165,E2 1234.165} C_VEL
LIN {X 0,Y 345.05,Z 816.252,A -85,B 0,C 180,E1 1234.051,E2 1234.051} C_VEL
LIN {X 0,Y 344.022,Z 813.794,A -85,B 0,C 180,E1 1230.345,E2 1230.345} C_VEL
LIN {X 0,Y 343.296,Z 813.308,A -85,B 0,C 180,E1 1224.985,E2 1224.985} C_VEL
LIN {X 0,Y 344.034,Z 813.602,A -85,B 0,C 180,E1 1220.022,E2 1220.022} C_VEL
LIN {X 0,Y 343.874,Z 814.589,A -85,B 0,C 180,E1 1219.804,E2 1219.804} C_VEL
LIN {X 0,Y 343.229,Z 817.624,A -85,B 0,C 180,E1 1219.724,E2 1219.724} C_VEL
LIN {X 0,Y 342.176,Z 822.197,A -85,B 0,C 180,E1 1219.93,E2 1219.93} C_VEL
LIN {X 0,Y 339.831,Z 831.843,A -85,B 0,C 180,E1 1220.7,E2 1220.7} C_VEL
LIN {X 0,Y 338.653,Z 836.487,A -85,B 0,C 180,E1 1220.833,E2 1220.833} C_VEL
LIN {X 0,Y 331.105,Z 863.942,A -85,B 0,C 180,E1 1220.759,E2 1220.759} C_VEL
LIN {X 0,Y 321.831,Z 892.133,A -85,B 0,C 180,E1 1220.679,E2 1220.679} C_VEL
LIN {X 0,Y 310.812,Z 919.727,A -85,B 0,C 180,E1 1220.597,E2 1220.597} C_VEL
LIN {X 0,Y 299.58,Z 944.257,A -85,B 0,C 180,E1 1220.525,E2 1220.525} C_VEL
LIN {X 0,Y 285.26,Z 971.352,A -85,B 0,C 180,E1 1220.455,E2 1220.455} C_VEL
LIN {X 0,Y 271.967,Z 993.49,A -85,B 0,C 180,E1 1220.415,E2 1220.415} C_VEL
LIN {X 0,Y 255.66,Z 1017.804,A -85,B 0,C 180,E1 1220.395,E2 1220.395} C_VEL
LIN {X 0,Y 238.484,Z 1040.225,A -85,B 0,C 180,E1 1220.41,E2 1220.41} C_VEL
LIN {X 0,Y 222.976,Z 1058.553,A -85,B 0,C 180,E1 1220.47,E2 1220.47} C_VEL
LIN {X 0,Y 203.105,Z 1079.721,A -85,B 0,C 180,E1 1220.615,E2 1220.615} C_VEL
LIN {X 0,Y 183.764,Z 1097.919,A -85,B 0,C 180,E1 1220.863,E2 1220.863} C_VEL
LIN {X 0,Y 165.408,Z 1113.5,A -85,B 0,C 180,E1 1221.242,E2 1221.242} C_VEL
LIN {X 0,Y 142.847,Z 1130.756,A -85,B 0,C 180,E1 1221.977,E2 1221.977} C_VEL
LIN {X 0,Y 121.281,Z 1145.206,A -85,B 0,C 180,E1 1223.101,E2 1223.101} C_VEL
LIN {X 0,Y 101.602,Z 1157.119,A -85,B 0,C 180,E1 1224.767,E2 1224.767} C_VEL
LIN {X 0,Y 101.118,Z 1157.411,A -85,B 0,C 180,E1 1224.872,E2 1224.872} C_VEL
LIN {X 0,Y 118.596,Z 1147.757,A -85,B 0,C 180,E1 1226.581,E2 1226.581} C_VEL
LIN {X 0,Y 138.068,Z 1135.668,A -85,B 0,C 180,E1 1227.919,E2 1227.919} C_VEL
LIN {X 0,Y 162.019,Z 1118.694,A -85,B 0,C 180,E1 1229.073,E2 1229.073} C_VEL
LIN {X 0,Y 180.583,Z 1103.706,A -85,B 0,C 180,E1 1229.743,E2 1229.743} C_VEL
LIN {X 0,Y 198.072,Z 1088.052,A -85,B 0,C 180,E1 1230.257,E2 1230.257} C_VEL
LIN {X 0,Y 218.071,Z 1068.102,A -85,B 0,C 180,E1 1230.742,E2 1230.742} C_VEL
LIN {X 0,Y 236.074,Z 1047.662,A -85,B 0,C 180,E1 1231.128,E2 1231.128} C_VEL
LIN {X 0,Y 251.63,Z 1028.062,A -85,B 0,C 180,E1 1231.422,E2 1231.422} C_VEL
LIN {X 0,Y 269.665,Z 1002.384,A -85,B 0,C 180,E1 1231.762,E2 1231.762} C_VEL
LIN {X 0,Y 283.071,Z 980.691,A -85,B 0,C 180,E1 1232.014,E2 1232.014} C_VEL
LIN {X 0,Y 297.042,Z 955.337,A -85,B 0,C 180,E1 1232.287,E2 1232.287} C_VEL
LIN {X 0,Y 309.478,Z 928.955,A -85,B 0,C 180,E1 1232.549,E2 1232.549} C_VEL
LIN {X 0,Y 319.42,Z 904.828,A -85,B 0,C 180,E1 1232.748,E2 1232.748} C_VEL
LIN {X 0,Y 329.645,Z 875.187,A -85,B 0,C 180,E1 1232.834,E2 1232.834} C_VEL
LIN {X 0,Y 336.702,Z 850.288,A -85,B 0,C 180,E1 1232.818,E2 1232.818} C_VEL
LIN {X 0,Y 342.972,Z 823.255,A -85,B 0,C 180,E1 1232.737,E2 1232.737} C_VEL
LIN {X 0,Y 342.376,Z 821.605,A -85,B 0,C 180,E1 1230.153,E2 1230.153} C_VEL
LIN {X 0,Y 341.658,Z 821.131,A -85,B 0,C 180,E1 1224.792,E2 1224.792} C_VEL
LIN {X 0,Y 342.043,Z 821.477,A -85,B 0,C 180,E1 1220.874,E2 1220.874} C_VEL
LIN {X 0,Y 338.653,Z 836.487,A -85,B 0,C 180,E1 1220.833,E2 1220.833} C_VEL
LIN {X 0,Y 336.704,Z 843.94,A -85,B 0,C 180,E1 1220.994,E2 1220.994} C_VEL
LIN {X 0,Y 331.365,Z 862.481,A -85,B 0,C 180,E1 1221.985,E2 1221.985} C_VEL
LIN {X 0,Y 329.106,Z 869.871,A -85,B 0,C 180,E1 1222.133,E2 1222.133} C_VEL
LIN {X 0,Y 318.985,Z 899.156,A -85,B 0,C 180,E1 1222.093,E2 1222.093} C_VEL
LIN {X 0,Y 309.066,Z 923.531,A -85,B 0,C 180,E1 1222.07,E2 1222.07} C_VEL
LIN {X 0,Y 296.195,Z 951.021,A -85,B 0,C 180,E1 1222.059,E2 1222.059} C_VEL
LIN {X 0,Y 283.026,Z 975.284,A -85,B 0,C 180,E1 1222.068,E2 1222.068} C_VEL
LIN {X 0,Y 269.173,Z 998.076,A -85,B 0,C 180,E1 1222.112,E2 1222.112} C_VEL
LIN {X 0,Y 251.326,Z 1023.913,A -85,B 0,C 180,E1 1222.216,E2 1222.216} C_VEL
LIN {X 0,Y 236.134,Z 1043.482,A -85,B 0,C 180,E1 1222.356,E2 1222.356} C_VEL
LIN {X 0,Y 217.352,Z 1065.315,A -85,B 0,C 180,E1 1222.609,E2 1222.609} C_VEL
LIN {X 0,Y 197.703,Z 1085.398,A -85,B 0,C 180,E1 1222.997,E2 1222.997} C_VEL
LIN {X 0,Y 180.424,Z 1101.412,A -85,B 0,C 180,E1 1223.472,E2 1223.472} C_VEL
LIN {X 0,Y 158.778,Z 1119.596,A -85,B 0,C 180,E1 1224.327,E2 1224.327} C_VEL
LIN {X 0,Y 144.721,Z 1130.219,A -85,B 0,C 180,E1 1225.13,E2 1225.13} C_VEL
LIN {X 0,Y 164.456,Z 1115.74,A -85,B 0,C 180,E1 1226.403,E2 1226.403} C_VEL
LIN {X 0,Y 181.826,Z 1101.542,A -85,B 0,C 180,E1 1227.284,E2 1227.284} C_VEL
LIN {X 0,Y 200.329,Z 1084.78,A -85,B 0,C 180,E1 1228.049,E2 1228.049} C_VEL
LIN {X 0,Y 221.035,Z 1063.555,A -85,B 0,C 180,E1 1228.756,E2 1228.756} C_VEL
LIN {X 0,Y 237.354,Z 1044.782,A -85,B 0,C 180,E1 1229.246,E2 1229.246} C_VEL
LIN {X 0,Y 254.769,Z 1022.531,A -85,B 0,C 180,E1 1229.703,E2 1229.703} C_VEL
LIN {X 0,Y 271.001,Z 998.785,A -85,B 0,C 180,E1 1230.117,E2 1230.117} C_VEL
LIN {X 0,Y 284.471,Z 976.774,A -85,B 0,C 180,E1 1230.45,E2 1230.45} C_VEL
LIN {X 0,Y 299.476,Z 948.733,A -85,B 0,C 180,E1 1230.826,E2 1230.826} C_VEL
LIN {X 0,Y 310.608,Z 924.758,A -85,B 0,C 180,E1 1231.115,E2 1231.115} C_VEL
LIN {X 0,Y 321.553,Z 897.45,A -85,B 0,C 180,E1 1231.362,E2 1231.362} C_VEL
LIN {X 0,Y 330.366,Z 870.833,A -85,B 0,C 180,E1 1231.454,E2 1231.454} C_VEL
LIN {X 0,Y 337.742,Z 844.179,A -85,B 0,C 180,E1 1231.453,E2 1231.453} C_VEL
LIN {X 0,Y 340.94,Z 830.173,A -85,B 0,C 180,E1 1231.416,E2 1231.416} C_VEL
LIN {X 0,Y 340.559,Z 829.37,A -85,B 0,C 180,E1 1229.863,E2 1229.863} C_VEL
LIN {X 0,Y 339.959,Z 828.932,A -85,B 0,C 180,E1 1224.383,E2 1224.383} C_VEL
LIN {X 0,Y 340.081,Z 829.147,A -85,B 0,C 180,E1 1222.2,E2 1222.2} C_VEL
LIN {X 0,Y 331.744,Z 861.108,A -85,B 0,C 180,E1 1222.147,E2 1222.147} C_VEL
LIN {X 0,Y 329.106,Z 869.871,A -85,B 0,C 180,E1 1222.133,E2 1222.133} C_VEL
LIN {X 0,Y 326.456,Z 878.252,A -85,B 0,C 180,E1 1222.341,E2 1222.341} C_VEL
LIN {X 0,Y 320.103,Z 896.399,A -85,B 0,C 180,E1 1223.409,E2 1223.409} C_VEL
LIN {X 0,Y 317.691,Z 902.584,A -85,B 0,C 180,E1 1223.532,E2 1223.532} C_VEL
LIN {X 0,Y 307.335,Z 927.666,A -85,B 0,C 180,E1 1223.56,E2 1223.56} C_VEL
LIN {X 0,Y 293.868,Z 955.671,A -85,B 0,C 180,E1 1223.621,E2 1223.621} C_VEL
LIN {X 0,Y 281.618,Z 977.981,A -85,B 0,C 180,E1 1223.703,E2 1223.703} C_VEL
LIN {X 0,Y 266.127,Z 1003.157,A -85,B 0,C 180,E1 1223.851,E2 1223.851} C_VEL
LIN {X 0,Y 250.073,Z 1025.964,A -85,B 0,C 180,E1 1224.063,E2 1224.063} C_VEL
LIN {X 0,Y 234.896,Z 1045.461,A -85,B 0,C 180,E1 1224.326,E2 1224.326} C_VEL
LIN {X 0,Y 215.416,Z 1067.964,A -85,B 0,C 180,E1 1224.778,E2 1224.778} C_VEL
LIN {X 0,Y 196.88,Z 1086.936,A -85,B 0,C 180,E1 1225.359,E2 1225.359} C_VEL
LIN {X 0,Y 194.199,Z 1089.544,A -85,B 0,C 180,E1 1225.466,E2 1225.466} C_VEL
LIN {X 0,Y 210.587,Z 1073.591,A -85,B 0,C 180,E1 1226.253,E2 1226.253} C_VEL
LIN {X 0,Y 227.807,Z 1055.079,A -85,B 0,C 180,E1 1226.964,E2 1226.964} C_VEL
LIN {X 0,Y 246.641,Z 1032.12,A -85,B 0,C 180,E1 1227.647,E2 1227.647} C_VEL
LIN {X 0,Y 261.413,Z 1011.927,A -85,B 0,C 180,E1 1228.14,E2 1228.14} C_VEL
LIN {X 0,Y 277.509,Z 987.341,A -85,B 0,C 180,E1 1228.641,E2 1228.641} C_VEL
LIN {X 0,Y 291.415,Z 962.901,A -85,B 0,C 180,E1 1229.068,E2 1229.068} C_VEL
LIN {X 0,Y 303.113,Z 939.764,A -85,B 0,C 180,E1 1229.424,E2 1229.424} C_VEL
LIN {X 0,Y 315.403,Z 911.627,A -85,B 0,C 180,E1 1229.803,E2 1229.803} C_VEL
LIN {X 0,Y 323.904,Z 888.858,A -85,B 0,C 180,E1 1229.994,E2 1229.994} C_VEL
LIN {X 0,Y 332.225,Z 862.8,A -85,B 0,C 180,E1 1230.086,E2 1230.086} C_VEL
LIN {X 0,Y 338.896,Z 837.218,A -85,B 0,C 180,E1 1230.091,E2 1230.091} C_VEL
LIN {X 0,Y 338.205,Z 836.754,A -85,B 0,C 180,E1 1224.794,E2 1224.794} C_VEL
LIN {X 0,Y 338.23,Z 836.979,A -85,B 0,C 180,E1 1223.54,E2 1223.54} C_VEL
LIN {X 0,Y 330.444,Z 865.347,A -85,B 0,C 180,E1 1223.528,E2 1223.528} C_VEL
LIN {X 0,Y 321.284,Z 893.187,A -85,B 0,C 180,E1 1223.528,E2 1223.528} C_VEL
LIN {X 0,Y 317.691,Z 902.584,A -85,B 0,C 180,E1 1223.532,E2 1223.532} C_VEL
LIN {X 0,Y 314.913,Z 909.758,A -85,B 0,C 180,E1 1223.724,E2 1223.724} C_VEL
LIN {X 0,Y 307.168,Z 928.467,A -85,B 0,C 180,E1 1224.913,E2 1224.913} C_VEL
LIN {X 0,Y 304.407,Z 934.466,A -85,B 0,C 180,E1 1225.073,E2 1225.073} C_VEL
LIN {X 0,Y 291.846,Z 959.887,A -85,B 0,C 180,E1 1225.205,E2 1225.205} C_VEL
LIN {X 0,Y 278.63,Z 983.635,A -85,B 0,C 180,E1 1225.378,E2 1225.378} C_VEL
LIN {X 0,Y 262.279,Z 1009.374,A -85,B 0,C 180,E1 1225.651,E2 1225.651} C_VEL
LIN {X 0,Y 249.713,Z 1027.157,A -85,B 0,C 180,E1 1225.93,E2 1225.93} C_VEL
LIN {X 0,Y 266.513,Z 1003.664,A -85,B 0,C 180,E1 1226.59,E2 1226.59} C_VEL
LIN {X 0,Y 281.494,Z 979.637,A -85,B 0,C 180,E1 1227.146,E2 1227.146} C_VEL
LIN {X 0,Y 293.99,Z 957.096,A -85,B 0,C 180,E1 1227.599,E2 1227.599} C_VEL
LIN {X 0,Y 307.457,Z 929.186,A -85,B 0,C 180,E1 1228.081,E2 1228.081} C_VEL
LIN {X 0,Y 317.191,Z 905.816,A -85,B 0,C 180,E1 1228.42,E2 1228.42} C_VEL
LIN {X 0,Y 326.232,Z 880.773,A -85,B 0,C 180,E1 1228.63,E2 1228.63} C_VEL
LIN {X 0,Y 334.807,Z 851.82,A -85,B 0,C 180,E1 1228.73,E2 1228.73} C_VEL
LIN {X 0,Y 336.641,Z 844.812,A -85,B 0,C 180,E1 1228.737,E2 1228.737} C_VEL
LIN {X 0,Y 336.141,Z 844.694,A -85,B 0,C 180,E1 1224.902,E2 1224.902} C_VEL
LIN {X 0,Y 328.818,Z 870.572,A -85,B 0,C 180,E1 1224.919,E2 1224.919} C_VEL
LIN {X 0,Y 318.393,Z 900.855,A -85,B 0,C 180,E1 1224.97,E2 1224.97} C_VEL
LIN {X 0,Y 308.665,Z 924.78,A -85,B 0,C 180,E1 1225.041,E2 1225.041} C_VEL
